FUNCTION "GCS7_SecCtrlMain" : VOID	// FC 60
TITLE = Section Control: Main function
//COPYRIGHT:    (C) 1994 BY  BUHLER AG,  CH-9240 UZWIL  SWITZERLAND
//
//PRODUCT:      GCS7
//
//TITLE:        SECTION CONTROL: MAIN PROGRAM
//
//-------------------------------------------------------------------------
//
//IDENT:        AUTOR:              DEPT:                         DATE:
//
//FB60.3.7      A.Egli              CT3                           07-Mar-2005
//              Move Data: StErrBatch is bit DBX201.0 and not DBX165.0
//FB60.3.6      A.Egli              CT3                           27-Jan-2005
//              Move Data: Compare Job Number, don't use InfSameJobPrevSec 
//FB60.3.5      A.Egli              CT3                           12-Nov-2003
//              Transition to Active: Set JobAc.BatchNo=1 when < 0
//FB60.3.4      A.Egli              CT3                           04-Aug-2003
//              PCRead.Status.StaImmediateStopASW is DBX120.0
//FB60.3.3      A.Egli              CT3                           17-Jul-2003
//              PCDirectControl: ParLineNr is DBW2 and not DBW4
//FB60.3.2      A.Egli              CT3                           12-Jun-2003
//              Wrong lenght copy Line to section
//FB60.3.1      A.Egli              CT3                           14-Mar-2003
//              Code35: Move to any section DB: DBW20=Destination
//              Code22,23: No Transition StEmptying to StWait
//FB60.3.0      A.Egli              CT3                            8-Okt-2002
//              New release
//FB60.2.10     A.Egli              CT3                           18-Mar-2002
//  Send Command only to next section, if InfDataReady=1
//FB60.2.9      A.Egli              CT3                           24-Sept-2001
//  ParStartReleaseTime <=0 : Unlimited time
//FB60.2.8      A.Egli              CT3                           17-Mai-2001
//  Update Last Batch in next section
//FB60.2.7      A.Egli              CT3                            5-Jul-2000
//  Read command from PC only with F_Define 
//FB60.2.6      A.Egli              CT3                           13-Mar-2000
//  Replace DBB73 with DBW72 and DBB9 with DBW8 
//FB60.2E       A.Egli              CT3                           30-Apr-1999
// -Zustandswechsel nach st_emptied: Abfrage DBX117.3 nicht DIX117.3 
//FB60.2D       A.Egli              CT3                           01-Apr-1999
// -Methode 25: Move allways
// -Bei reset Zustandswechsel nach st_emptied (Verbuchung
// -Bei reset kein Zustandswechsel nach  StActive
//FB60.2C       A.Egli              CT3                           22-Jul-98
//               Line-Nr =DBW2
//FB60.2B       A.Egli              AEE6                          14-Mai-98
//               ToASW.InfDataMoved
//FB60.2A       A.Egli              AEE6                          14-Jan-98
//               Update  S5 (Version 2M)
//FB60.1A       A.Egli              AEE6                          16-Jun-96
//               Convert S5 to S7 (Version 2H)
//
//-------------------------------------------------------------------------
//
//PURPOSE:      MANUAL : GCSOSMAN
//
//RESTRICTIONS:
//
//-------------------------------------------------------------------------
//
// CODE of the Methode
//        0    : METHODE CONTROL
//        1    : METHODE DECODER
//        2    : METHODE STEP
//        3    : METHODE STEP_TRANSITION
//        4    : METHODE STATE
//        5    : METHODE MOVE_DATA
//        6    : METHODE NEXT BATCH
//        7    : METHODE O_SECTION
//        9    : METHODE ResultTotal
//        10   : METHODE ResultBatch
//        12   : METHODE PC Direct Control (Diagnose)
//        13   : METHODE WayAdJustTime  
//        25   : METHODE MOVE_DATA Uncondtion
//        35   : METHODE MOVE_DATA any section
//
//ACTUAL DB BY CALL: SECTION  DB
//AUFGESCHALGENER  : SEKTIONS DB
//
//$EJECT
//
//
//
//
//
AUTHOR : EA
FAMILY : GCS7UL
NAME : SEC_MAIN
VERSION : 3.7
VAR_INPUT
  CODE : INT ;	// CODE
END_VAR
VAR_TEMP
  Fault : BOOL ;
  VarLength : INT ;
  tmpByteWrite : INT ;
  SecDBAc : INT ;
  SecDBNext : INT ;
END_VAR
BEGIN
NETWORK
TITLE =
      L     DBNO;
      T     #SecDBAc;
NETWORK
TITLE =  METHODE CONTROL
      L     #CODE;
      L     0;
      <>I;
      JC    aEnd;
// === COMMANDS ==================
      L     DBD 46;	// "SecDB".ToASW.Func
      L     DBD 66;	// "SecDB".ToSSW.Func
      OD;	// 
      T     DBD 46;	// ->"SecDB".ToASW.Func
      L     0;	// 
      ==D;	//   no new commands
      JC    aNoC;
//=== RESET STATUSBIT ======
      L     2#111111;	// ON-COMMAND
      L     DBW 46;	// "SecDB".ToASW.Func[31..16]
      AW;	// 
      INVI;	// 
      L     DBW 120;	// "SecDB".PCRead.Status[15..00]
      AW;	// 
      T     DBW 120;	// ->"SecDB".PCRead.Status[15..00]
// === SET STATUSBIT  ======
      L     2#11111111;	// OFF-COMMAND
      L     DBW 48;	// "SecDB".ToASW.Func[15..00]
      AW;	// 
      L     DBW 120;	// "SecDB".PCRead.Status[15..00]
      OW;	// 
      T     DBW 120;	// -->"SecDB".PCRead.StatusS[15..00]
// 
      A     DBX 121.6;	// "SecDB".PCRead.Status.StaReset
      S     DBX 121.7;	//  "SecDB".PCRead.Status.StaEndOfJob
      A     DBX 48.1;	// "SecDB".ToASW.Func.CmdAbortBacth
      S     DBX 201.0;	// ->"SecDB".JobAc.StaBatch.StaErrBatch
      A     DBX 49.6;	// "SecDB".ToASW.Func.CmdReset
      O     DBX 49.7;	// "SecDB".ToASW.Func.CmdSequenzStop
      O     DBX 48.1;	// "SecDB".ToASW.Func.CmdAbortBacth
      A     DBX 45.7;	//"SecDB".ToASW.InfDataReady [2.10]
      JCN   aNoC;
      CALL  "GCS7_SecCtrlSub" (
           CODE                     := 2);	// SUBROUTINE SEQUENZ_STOP
aNoC: L     0;	// 
      T     DBD 66;	// -> "SecDB".ToSSW.Func
      L     DBW 206;	// "SecDB".JobAc.BatchNo
      L     DBW 168;	// "SecDB".JobNom.BatchNo
      >=I;	// 
      S     DBX 201.3;	// -> "SecDB".JobAc.StaBatch.StaLastBatch
      CALL  "GCS7_SecCtrlSub" (
           CODE                     := 1);	// SUBROUTINE compare
//===Empyting Time =====================================
      AN    DBX 64.2;	//"SecDB".ToSSW.InfPulseTimer
      O     DBX 45.0;	//  "SecDB".ToASW.InfEmptyingTimeEnd
      JC    aE2;	// 
      L     DBW 132;	//"SecDB".PCRead.OutEmptyingTime
      +     1;	// 
      T     DBW 132;	// ->"SecDB".PCRead.OutEmptyingTime
// 
aE2:  A     DBX 62.5;	// "SecDB".ToSSW.InfFeeding
      S     DBX 119.4;	// ->"SecDB".PCRead.Status.StaLoaded
      A     DBX 64.7;	// "SecDB".ToSSW.InfReleaseEmptyingTime
      JC    aX3;	// 
      L     0;	// 
      T     DBW 132;	// "SecDB".PCRead.OutEmptyingTime
aX3:  L     DBW 100;	// "SecDB".PCWrite.ParEmptyingTime
      L     DBW 132;	// "SecDB".PCRead.OutEmptyingTime
      <=I;	// 
      A     DBX 64.7;	//"SecDB".ToSSW.InfReleaseEmptyingTime 
      =     DBX 45.0;	//"SecDB".ToASW.InfEmptyingTimeEnd
      R     DBX 119.4;	// ->"SecDB".PCRead.Status.StaLoaded
      AN    DBX 45.0;	//"SecDB".ToASW.InfEmptyingTimeEnd
      A     DBX 64.7;	// "SecDB".ToSSW.InfReleaseEmptyingTime
      =     DBX 119.6;	// -> "SecDB".PCRead.Status.StaEmptyingTime
//===== F_RESULT =================
      AN    DBX 64.1;	// "SecDB".ToSSW.CmdSendResult
      JC    aCMD;	// 
      AN    DBX 82.1;	// "SecDB".PCWrite.Hsk.Q_Result
      AN    DBX 201.2;	// "SecDB".JobAc.StaBatch.StaRegistrated
      AN    DBX 102.1;	//  "SecDB".PCRead.Hsk.F_Result
      S     DBX 102.1;	//  "SecDB".PCRead.Hsk.F_Result
      S     DBX 41.0;	//  "SecDB".ChangeBit.CBit1 
aCMD: BEU;
aEnd: NOP   0;
NETWORK
TITLE =  METHODE DECODER (Code 1)
      L     #CODE;
      L     1;
      <>I;
      JC    bEnd;
      L     0;
      L     DBB 145;	//  "LineDB".JobWrite.Hsk
      ==I;
      BEC;
      L     DBW 140;	// "LineDB".JobRead.ErrCode   [*1C*]
      L     0;
      <>I;
      BEC;
      L     64;	// Job-Header
      T     DBW 20;	// "LineDB".VarTemp[1] = ObjectNr
      CALL  "GCS7_LineCtrlSub" (
           CODE                     := 1);	// Subroutine block_adr
      OPN   DI [DBW 4];	// -->CALL SECTION-DB[ "LineDB".Para.ParFirstSecDB]
bLop: AN    DIX 44.7;	// "SecDB".ToASW.InfSameJobLineDB
      JC    bNxt;
//  ==== modify datas ===========
      S     DIX 44.0;	// "SecDB".ToASW.CmdModify  
      L     DBD 156;	// "LineDB".JobWrite.Func
      L     DID 46;	// "SecDB".ToASW.Func
      OD;	// 
      T     DID 46;	// --> "SecDB".ToASW.Func
// === Job-Header ==========
      L     DINO;
      T     #SecDBAc;
      CALL  "SYS_Copy_DBtoDB" (
           DBSource                 := DIW 4,
           ByteSource               := 160,
           DBDest                   := #SecDBAc,
           ByteDest                 := 160,
           NoOfByte                 := 40,
           Fault                    := #Fault);	//L_DB / L_DB.DBB160 / SecDB / SecDB.DBB160
// === Telegram: Additional data===
      L     DBW 22;	// "LineDB".VarTemp[2]= VarDWNr
      L     0;	// 
      ==I;	// 
      JC    bEXE;	// 
      L     DIW 12;	// "SecDB".Para.ParSecDataLenNomValue
      T     #VarLength;	// ->VarLenth
      L     DIW 10;	// "SecDB".Para.ParSecDataFirstByte
      L     DIW 14;	// "SecDB".Para.ParSecDataLenAcValue [3.1]
      +I;
      T     #tmpByteWrite;
      CALL  "SYS_Copy_DBtoDB" (
           DBSource                 := DIW 4,
           ByteSource               := DBW 22,
           DBDest                   := #SecDBAc,
           ByteDest                 := #tmpByteWrite,
           NoOfByte                 := #VarLength,
           Fault                    := #Fault);	//L_DB / L_DB.VarDWNr / SecDB
bEXE: AN    DBX 145.1;	//"LineDB".JobWrite.Hsk.F_Execute
      JC    bNxt;
      R     DBX 153.7;	// "LineDB".JobWrite.ObjMask[64]
      L     DBD 146;	// "LineDB".JobWrite.ObjMask[64..01]
      L     DBD 150;	// "LineDB".JobWrite.ObjMask[64..01]
      OD;
      JN    bNxt;
      CDB;
      CALL  "GCS7_SecCtrlSub" (
           CODE                     := 3);	// SUBROUTINE init_section
      CDB;
// -- Call next section
bNxt: L     DIW 8;	// "SecDB".Para.ParNextSecDB
      L     0;	//  
      ==I;	// no next section
      JC    bINI;	// 
      OPN   DI [DIW 8];	// ->CALL SECTION-DB["SecDB".Para.ParNextSecDB]
      JU    bLop;
bINI: R     DBX 153.7;	// "LineDB".JobWrite.ObjMask[64]
      BEU;
bEnd: NOP   0;
NETWORK
TITLE =  METHODE STEP (Code 2 , 22) 
      L     #CODE;
      L     2;
      <>I;
      A(;
      L     #CODE;
      L     22;
      <>I;
      );
      JC    cEnd;
      L     0;
      T     DBW 50;	// "SecDB".ToASW.Transition:=0
      A     DBX 111.0;	//"SecDB".PCRead.Step.StPassive
      JC    cS0;
      A     DBX 111.1;	// "SecDB".PCRead.Step.StWait
      JC    cS1;	// 
      A     DBX 111.2;	//  "SecDB".PCRead.Step.StActive
      JC    cS2;
      A     DBX 111.3;	//  "SecDB".PCRead.Step.StReady
      JC    cS3;
      A     DBX 111.4;	//  "SecDB".PCRead.Step.StEmptying
      JC    cS4;
      A     DBX 111.5;	//  "SecDB".PCRead.Step.StEmptied
      JC    cS5;
      A     DBX 111.6;	//  "SecDB".PCRead.Step.StIdling
      JC    cS6;
      S     DBX 111.0;	// "SecDB".PCRead.Step.StPassive
// === ST_PASSIVE  ========================================
cS0:  A     DBX 45.7;	//"SecDB".ToASW.InfDataReady
      JC    cTx1;	// --> StWait
      JU    cEnd;
// === ST_WAIT ============================================
cS1:  A(;
      L     #CODE;
      L     2;
      ==I;
      );
      A     DBX 121.7;	// "SecDB".PCRead.Status.StaEndOfJob
      AN    DBX 44.5;	// "SecDB".ToASW.InfSameBatchPrevSec
      O     DBX 121.6;	// "SecDB".PCRead.Status.StaReset
      ON    DBX 45.7;	// "SecDB".ToASW.InfDataReady
      JC    cTx5;	// --> StEmpting [2D]
      AN    DBX 116.0;	// es_batchSize
      A     DBX 63.1;	// "SecDB".ToSSW.CmdGotoActive
      JC    cTx2;	// -->  "SecDB".PCRead.Step.StActive
      JU    cEnd;
// ===  "SecDB".PCRead.Step.StActive ==========================================
cS2:  A     DBX 63.2;	// "SecDB".ToSSW.CmdGotoReady
      AN    DBX 44.5;	// "SecDB".ToASW.InfSameBatchPrevSec
      JC    cTx3;	// -->  "SecDB".PCRead.Step.StReady
      L     DBW 72;	//  "SecDB".ToSSW.InNextSecDB
      L     0;	// 
      ==I;	// 
      O     DBX 44.6;	// "SecDB".ToASW.InfSameBatchNextSec
      AN    DBX 44.5;	// "SecDB".ToASW.InfSameBatchPrevSec
      A     DBX 63.3;	//"SecDB".ToSSW.CmdGotoEmptying
      JC    cTx4;	// 
      A     DBX 121.6;	// "SecDB".PCRead.Status.StaReset
      ON    DBX 45.7;	// "SecDB".ToASW.InfDataReady
      JC    cTx5;	// --> StEmpting [2D]
      JU    cEnd;
// ===  "SecDB".PCRead.Step.StReady ==========================================
cS3:  L     DBW 72;	// "SecDB".ToSSW.InNextSecDB
      L     0;	// 
      ==I;	// 
      O     DBX 44.6;	// "SecDB".ToASW.InfSameBatchNextSec
      A     DBX 63.3;	// "SecDB".ToSSW.CmdGotoEmptying
      JC    cTx4;	// -->  "SecDB".PCRead.Step.StEmptying
      A     DBX 121.6;	//  "SecDB".PCRead.Status.StaReset
      ON    DBX 45.7;	//"SecDB".ToASW.InfDataReady
      JC    cTx5;	// --> StEmpting [2D]
      JU    cEnd;
// ===  "SecDB".PCRead.Step.StEmptying =======================================
cS4:  A     DBX 44.5;	// "SecDB".ToASW.InfSameBatchPrevSec
      JC    cTx2;	// -->  "SecDB".PCRead.Step.StActive
      L     DBW 72;	//  "SecDB".ToSSW.InNextSecDB
      L     0;	// 
      ==I;	// 
      O     DBX 44.6;	// "SecDB".ToASW.InfSameBatchNextSec
      A     DBX 63.4;	// "SecDB".ToSSW.CmdGotoEmptied
      JC    cTx5;	// --> StEmptied
      A     DBX 121.6;	//  "SecDB".PCRead.Status.StaReset
      ON    DBX 45.7;	// "SecDB".ToASW.InfDataReady 
      JC    cTx5;	// --> StEmpting [2D]
      JU    cEnd;
// === ST_EMPTIED =======================================
cS5:  A     DBX 44.5;	// "SecDB".ToASW.InfSameBatchPrevSec
      AN    DBX 121.6;	// STA_RESET  [2D]
      JC    cTx2;	// -->  "SecDB".PCRead.Step.StActive
      L     DBW 206;	// "SecDB".JobAc.BatchNo 
      L     DBW 168;	// "SecDB".JobNom.BatchNo
      >=I;	// 
      S     DBX 121.7;	// --> "SecDB".PCRead.Status.StaEndOfJob
      L     0;	// 
      L     DBW 70;	// "SecDB".ToSSW.InPrevSecDB
      ==I;	// 
      A(;
      L     #CODE;
      L     22;
      <>I;
      );
      AN    DBX 121.6;	// "SecDB".PCRead.Status.StaReset 
      AN    DBX 121.7;	// "SecDB".PCRead.Status.StaEndOfJob
      A     DBX 45.7;	// "SecDB".ToASW.InfDataReady
      A     DBX 63.5;	// "SecDB".ToSSW.CmdGotoIdling
      JC    cTx1;	// -->StWait
      A     DBX 121.6;	// "SecDB".PCRead.Status.StaReset [2D]
      ON    DBX 45.7;	//  "SecDB".ToASW.InfDataReady
      AN    DBX 119.3;	//"SecDB".PCRead.Status.StaOnline [2E]
      O     DBX 63.5;	// "SecDB".ToSSW.CmdGotoIdling
      JC    cTx6;	// ->  "SecDB".PCRead.Step.StIdling
      JU    cEnd;
// ===  "SecDB".PCRead.Step.StIdling =======================================
cS6:  A     DBX 45.7;	//  "SecDB".ToASW.InfDataReady
      JC    cTx1;	// --> StWait
      A     DBX 63.6;	//  "SecDB".ToSSW.CmdGotoPassive
      JC    cTx0;	// --> StPassive
      JU    cEnd;
// === TRANSITION =======================================
cTx0: L     2#1;	// --> "SecDB".PCRead.Step.StPassive
      JU    cTra;	// 
cTx1: L     2#10;	// --> "SecDB".PCRead.Step.StWait
      JU    cTra;	// 
cTx2: L     2#100;	// --> "SecDB".PCRead.Step.StActive
      JU    cTra;	// 
cTx3: L     2#1000;	// --> "SecDB".PCRead.Step.StReady
      JU    cTra;	// 
cTx4: L     2#10000;	// --> "SecDB".PCRead.Step.StEmptying
      JU    cTra;	// 
cTx5: L     2#100000;	// --> "SecDB".PCRead.Step.Emptied
      JU    cTra;	// 
cTx6: L     2#1000000;	// -->  "SecDB".PCRead.Step.StIdling
// ==== ALL TRANSITION ==================================
cTra: T     DBW 50;	// --> "SecDB".ToASW.Transition
      BEU;
cEnd: NOP   0;
NETWORK
TITLE =  METHODE TRANSITION_STEP (code 3)
      L     #CODE;
      L     3;
      <>I;
      A(;
      L     #CODE;
      L     23;
      <>I;
      );
      JC    dEnd;
      L     DBW 50;	// "SecDB".ToASW.Transition
      L     0;	// 
      ==I;	// 
      BEC;	// EXIT
      A     DBX 51.0;	// "SecDB".ToASW.Transition.ToPassive
      JC    dTx0;
      A     DBX 51.1;	// "SecDB".ToASW.Transition.ToWait
      JC    dTx1;
      A     DBX 51.2;	// "SecDB".ToASW.Transition.ToActive 
      JC    dTx2;
      A     DBX 51.3;	// "SecDB".ToASW.Transition.ToReady
      JC    dTx3;
      A     DBX 51.4;	// "SecDB".ToASW.Transition.ToEmptying
      JC    dTx4;
      A     DBX 51.5;	// "SecDB".ToASW.Transition.ToEmptied 
      JC    dTx5;
      A     DBX 51.6;	//"SecDB".ToASW.Transition.ToIdling
      JC    dTx6;
      JU    dEnd;
// === TRANSITION_TO_ST_PASSIVE =========================
dTx0: NOP   0;
      JU    dTra;
// === TRANSITION_TO_ST_WAIT ============================
dTx1: R     DBX 63.1;	//  "SecDB".ToSSW.CmdGotoActive 
      R     DBX 64.1;	// "SecDB".ToSSW.CmdSendResult
      A     DBX 111.5;	// "SecDB".PCRead.Step.StEmptied 
      R     DBX 201.0;	// -> "SecDB".JobAc.StaBatch.StaErrBatch
      JU    dTra;
// === TRANSITION_TO_ST_ACTIVE ==========================
dTx2: R     DBX 63.2;	// -> "SecDB".ToSSW.CmdGotoReady
      R     DBX 63.3;	// -> "SecDB".ToSSW.CmdGotoEmptying
      R     DBX 64.1;	// -> "SecDB".ToSSW.CmdSendResult
      L     DBW 206;	// "SecDB".JobAc.BatchNo  [3.5]
      L     1;	//                        [3.5]
      >=I;	//                        [3.5]
      ON    DBX 200.6;	// "SecDB".JobAc.StaBatch.StaEmptyingBatch [3.5]
      JC    dTra;	//                        [3.5]
      T     DBW 206;	// "SecDB".JobAc.BatchNo  [3.5]
      JU    dTra;
// === TRANSITION_TO_ST_READY ==========================
dTx3: R     DBX 63.3;	// -> "SecDB".ToSSW.CmdGotoEmptying
      JU    dTra;
// === TRANSITION_TO_ST_EMPYTYING ======================
dTx4: R     DBX 63.4;	// ->  "SecDB".ToSSW.CmdGotoEmptied
      JU    dTra;
// === TRANSITION_TO_ST_EMPYTIED =======================
dTx5: R     DBX 63.5;	// ->  "SecDB".ToSSW.CmdGotoIdling
      JU    dTra;
// === TRANSITION_TO_StIdling =========================
dTx6: R     DBX 63.6;	// -> "SecDB".ToSSW.CmdGotoPassive
      R     DBX 201.0;	// -> "SecDB".JobAc.StaBatch.StaErrBatch
      R     DBX 200.7;	// -> "SecDB".JobAc.StaBatch.StaScaleRecipeValid
      AN    DBX 121.7;	// [2.8]"SecDB".PCRead.Status.StaEndOfJob 
      JC    dT61;	// [2.8]                
      CALL  "GCS7_SecCtrlSub" (
           CODE                     := 2);	// [2.8] SUBROUTINE SEQUENZ_STOP
dT61: L     0;	// 
      L     DBW 70;	//  "SecDB".ToSSW.InPrevSecDB 
      <>I;	// 
      O(;
      L     #CODE;
      L     23;
      ==I;
      );
      O     DBX 121.7;	// "SecDB".PCRead.Status.StaEndOfJob
      R     DBX 45.7;	// -> "SecDB".ToASW.InfDataReady
      CALL  "GCS7_SecCtrlSub" (
           CODE                     := 7);	// Subroutine TestDone
      AN    DBX 39.0;	// OUTP.JobNotFound
      JC    dTra;	// 
      AN    DBX 102.0;	//  "SecDB".PCRead.Hsk.F_Status 
      S     DBX 201.4;	//"SecDB".JobAc.StaBatch.StaDone
      S     DBX 102.0;	// "SecDB".PCRead.Hsk.F_Status
      S     DBX 41.0;	// "SecDB".ChangeBit.CBit1
dTra: L     DBW 50;	//// "SecDB".ToASW.Transition
      T     DBB 111;	// -->"SecDB".PCRead.Step
      SET;	// 
      S     DBX 41.0;	//  "SecDB".ChangeBit.CBit1
      BEU;
dEnd: NOP   0;
NETWORK
TITLE =  METHODE STATE Code4
      L     #CODE;
      L     4;
      <>I;
      JC    eEnd;
      A     DBX 113.0;	// "SecDB".PCRead.State.StStopped
      JC    eS0;
      A     DBX 113.1;	// "SecDB".PCRead.State.StStarting
      JC    eS1;
      A     DBX 113.2;	// "SecDB".PCRead.State.StStarted 
      JC    eS2;
      A     DBX 113.3;	// "SecDB".PCRead.State.StStopping
      JC    eS3;
      A     DBX 113.5;	// "SecDB".PCRead.State.StFeeding
      JC    eS4;
      S     DBX 113.0;	// "SecDB".PCRead.State.StStopped
// === StStopped  ============
eS0:  AN    DBX 62.0;	// "SecDB".ToSSW.InfStopped
      JC    eT01;	// --> StStarting
      JU    eEnd;	// 
eT01: L     2#10;	// --> StStarting
      JU    eTra;
// === StStarting ============
eS1:  A     DBX 62.2;	// "SecDB".ToSSW.InfStarted
      JC    eT12;	// --> StStarted
      A     DBX 120.0;	// "SecDB".PCRead.Status.StaImmediateStopASW // [3.4]
      O     DBX 62.0;	// "SecDB".ToSSW.InfStopped
      O     DBX 111.6;	// "SecDB".PCRead.Step.StIdling
      JC    eT13;	// -> StStopping
      JU    eEnd;
eT12: L     2#100;	// -> StStarted
      JU    eTra;
eT13: L     2#1000;	// -> StStopping
      JU    eTra;
// === StStarted  ===========
eS2:  A     DBX 120.0;	// "SecDB".PCRead.Status.StaImmediateStopASW
      O     DBX 62.0;	// "SecDB".ToSSW.InfStopped
      JC    eT23;	// --> StStopping
      AN    DBX 62.2;	// "SecDB".ToSSW.InfStarted
      JC    eT21;	// --> StStarting
      A     DBX 62.5;	// "SecDB".ToSSW.InfFeeding
      JC    eT25;	// --> StFeeding
      JU    eEnd;
eT21: L     2#10;	// --> StStarting
      JU    eTra;
eT23: L     2#1000;	// --> StStopping
      JU    eTra;
eT25: L     2#100000;	// --> StFeeding
      JU    eTra;
// ==== STOPPING ==============
eS3:  A     DBX 62.0;	// "SecDB".ToSSW.InfStopped
      JC    eT30;	// -> StStopped
      AN    DBX 120.0;	// "SecDB".PCRead.Status.StaImmediateStopASW
      AN    DBX 62.0;	// "SecDB".ToSSW.InfStopped
      A     DBX 62.2;	// "SecDB".ToSSW.InfStarted
      JC    eT32;	// --> StStarted
      AN    DBX 120.0;	// "SecDB".PCRead.Status.StaImmediateStopASW
      AN    DBX 111.6;	// "SecDB".PCRead.Step.StIdling
      JC    eT32;	// --> StStarting
      JU    eEnd;
eT30: L     2#1;	// --> StStopped
      JU    eTra;
eT32: L     2#100;	// --> StStarted
      JU    eTra;
      L     2#10;	// --> StStarting
      JU    eTra;
// ==== FEEDING  ==============
eS4:  AN    DBX 62.5;	// "SecDB".ToSSW.InfFeeding
      JC    eT52;	// --> StStarted
      JU    eEnd;	// 
eT52: L     2#100;	// --> StStarted
// ==== ALL TRANSITION ========
eTra: T     DBB 113;	// --> "SecDB".PCRead.State
      SET;	// 
      S     DBX 41.0;	// Changebit.CBit1
      BEU;
eEnd: NOP   0;
NETWORK
TITLE =  METHODE MOVE_DATA Code 5,25,35
//Code 35:
//    Section destination=DBW20
      L     #CODE;
      L     5;
      ==I;
      JC    m5;
      L     #CODE;
      L     25;
      ==I;
      JC    m25;
      L     #CODE;
      L     35;
      <>I;
      JC    fEnd;
//Move to section DBW20
      R     DBX 44.2;	//S_DB[n].ToASW.CmdDataMoved
      L     0;
      L     DBW 20;	// "Sec".VarTemp.InOutValue1
      ==I;	// 
      BEC;	// --> no next section
      T     #SecDBNext;
      OPN   DI [#SecDBNext];	// >>>CALL NEXT SECTION-DB["SecDB".ToSSW.InNextSecDB]
      JU    m35;
//====== Move uncondition (Code=25)
m25:  R     DBX 44.2;	//S_DB[n].ToASW.CmdDataMoved
      L     DBW 72;	// "SecDB".ToSSW.InNextSecDB
      L     0;	// 
      ==I;	// 
      BEC;	// --> no next section
      AN    DBX 44.6;	//"SecDB".ToASW.InfSameBatchNextSec
      OPN   DI [DBW 72];	// >>>CALL NEXT SECTION-DB["SecDB".ToSSW.InNextSecDB]
      A     DIX 64.0;	// S_DB[n+1].ToSSW.InfReadyForNewBatch
      AN    DIX 121.3;	// S_DB[n+1].PCRead.Status.StaHold
      A(;
      AN    DIX 102.0;	// S_DB[n+1].PCRead.Hsk.F_Status
      ON    DIX 119.3;	// S_DB[n+1].PCRead.Status.StaOnline
      );
      JC    C3;
      BEU;	// THEN
//=== Move Regular (Code=5)
m5:   R     DBX 44.2;	//S_DB[n].ToASW.CmdDataMoved
      A     DBX 44.6;	// "SecDB".ToASW.InfSameBatchNextSec
      BEC;	//  
      L     DBW 72;	// "SecDB".ToSSW.InNextSecDB
      L     0;	// 
      ==I;	// 
      BEC;	// --> no next section
      OPN   DI [DBW 72];	// >>>CALL NEXT SECTION-DB["SecDB".ToSSW.InNextSecDB]
m35:  A     DBX 201.0;	// S_DB[n+1].JobAc.StaBatch.StaErrBatch
      A     DIX 45.7;	// S_DB[n+1].ToASW.InfDataRead
      BEC;	// 
      A     DIX 201.0;	// S_DB[n+1].JobAc.StaBatch.StaErrBatch       //[3.7]
      A     DIX 45.7;	// S_DB[n+1].ToASW.InfDataReady
      BEC;	// 
      A     DIX 111.0;	// S_DB[n+1].PCRead.Step.StPassive
      O     DIX 111.6;	// S_DB[n+1].PCRead.Step.StIdling
      O     DIX 111.4;	// S_DB[n+1].PCRead.Step.StEmptying
      O     DIX 111.5;	// S_DB[n+1].PCRead.Step.StEmptied
      JC    C2;
      BEU;	// THEN
C2:   A(;	// [3.6]
      L     DID 160;	// [3.6] S_DB[x].JobNom.JobNr
      L     DBD 160;	// [3.6] S_DB[n].JobNom.JobNr
      ==D;	// [3.6] --> InfSameJobPrevSec
      );	// [3.6]
      ON    DIX 45.7;	// S_DB[n+1].ToASW.InfDataReady
      A     DIX 64.0;	// S_DB[n+1].ToSSW.InfReadyForNewBatch
      AN    DIX 121.3;	// S_DB[n+1].PCRead.Status.StaHold
      A(;
      AN    DIX 102.0;	// S_DB[n+1].PCRead.Hsk.F_Status
      ON    DIX 119.3;	// S_DB[n+1].PCRead.Status.StaOnline
      );
      JC    C3;
      BEU;
// ==== MOVE DATA =================
// Copy header
C3:   L     DINO;
      T     #SecDBNext;
      CALL  "SYS_Copy_DBtoDB" (
           DBSource                 := #SecDBAc,
           ByteSource               := 160,
           DBDest                   := #SecDBNext,
           ByteDest                 := 160,
           NoOfByte                 := 80,
           Fault                    := #Fault);	//"SecDB".JobNom.JobNr / Sec[n+1].JobNom.JobNr
//-- copy dynamic datas 
      L     DIW 14;	//Para.ParSecDataLenAcValue
      L     DIW 12;	//Para.ParSecDataLenNomValue
      +I;
      T     #VarLength;
      CALL  "SYS_Copy_DBtoDB" (
           DBSource                 := #SecDBAc,
           ByteSource               := DBW 10,
           DBDest                   := #SecDBNext,
           ByteDest                 := DIW 10,
           NoOfByte                 := #VarLength,
           Fault                    := #Fault);	//Sec[n].Para.ParSecDataFirstByte / Sec[n+1].Para.ParSecDataFirstByte
//-- Copy bin data 
      CALL  "SYS_Copy_DBtoDB" (
           DBSource                 := #SecDBAc,
           ByteSource               := DBW 16,
           DBDest                   := #SecDBNext,
           ByteDest                 := DIW 16,
           NoOfByte                 := DIW 18,
           Fault                    := #Fault);	//Sec[n].Para.ParBinDataFirstByte / Sec[n+1].Para.ParBinDataFirstByte / Sec[n+1].Para.ParBinDataLength
// Init Sec[n+1]
      SET;
      S     DIX 45.7;	//S_DB[n+1].ToASW.InfDataReady 
      S     DIX 44.1;	//S_DB[n+1].ToASW.CmdNewBatch
      S     DBX 44.2;	//S_DB[n].ToASW.CmdDataMoved
      R     DIX 121.6;	//S_DB[n+1].PCRead.Status.StaReset
      R     DIX 121.7;	//S_DB[n+1].PCRead.Status.StaEndOfJob
      R     DIX 64.1;	//S_DB[n+1].ToSSW.CmdSendResult
      AN    DBX 121.0;	//S_DB[n].PCRead.Status.StaImmediateStop   
      R     DIX 121.0;	//S_DB[n+1].PCRead.Status.StaImmediateStop      
      AN    DBX 121.1;	//S_DB[n].PCRead.Status.StaTransferOff
      R     DIX 121.1;	//S_DB[n+1].PCRead.Status.StaTransferOff
      AN    DBX 121.2;	//S_DB[n].PCRead.Status.StaFeedOff
      R     DIX 121.2;	//S_DB[n+1].PCRead.Status.StaFeedOff
      CDB;	// 
      CALL  "GCS7_SecCtrlSub" (
           CODE                     := 1);	//SUBROUTINE compare S_DB[n+1]
      CDB;
      CALL  "GCS7_SecCtrlSub" (
           CODE                     := 1);	//SUBROUTINE compare S_DB[n]
      BEU;
fEnd: NOP   0;
NETWORK
TITLE =  METHODE NEXT_BATCH (code 6)
      L     #CODE;
      L     6;
      <>I;
      JC    gEnd;
      L     DBW 206;	// "SecDB".JobAc.BatchNo
      L     DBW 188;	// "SecDB".JobNom.BatchNoOffset
      >=I;
      JC    gOK;
      T     DBW 206;	// ->"SecDB".JobAc.BatchNo
gOK:  A     DBX 121.7;	// "SecDB".PCRead.Status.StaEndOfJob
      BEC;	// 
//==== start batch ===============
      CALL  "GCS7_SecCtrlSub" (
           CODE                     := 6);	// Subroutine CalcBatchSize
      A     DBX 116.0;	// "SecDB".PCRead.Fault.EsBatchSize
      O     DBX 121.7;	// "SecDB".PCRead.Status.StaEndOfJob
      BEC;
      L     DBD 210;	// "SecDB".JobAc.BatchWeightTarget
      L     DBD 202;	// "SecDB".JobAc.JobWeigth
      +D;	// 
      T     DBD 202;	// ->"SecDB".JobAc.JobWeigth
      L     DBW 206;	//  "SecDB".JobAc.BatchNo
      +     1;	// 
      T     DBW 206;	//  "SecDB".JobAc.BatchNo
      L     0;
      T     DBD 214;	// "SecDB".JobAc.BatchWeightActual
      SET;
      R     DBX 201.1;	//"SecDB".JobAc.StaBatch.StaHandAddReady
      R     DBX 201.2;	//"SecDB".JobAc.StaBatch.StaRegistrated
      L     DBW 206;	//"SecDB".JobAc.BatchNo
      L     DBW 168;	//"SecDB".JobNom.BatchNo
      >=I;	// 
      S     DBX 201.3;	//->"SecDB".JobAc.StaBatch.StaLastBatch 
      SET;	// 
      S     DBX 45.7;	//"SecDB".ToASW.InfDataReady
      S     DBX 44.1;	//"SecDB".ToASW.CmdNewBatch
      CALL  "GCS7_SecCtrlSub" (
           CODE                     := 1);	// SUBROUTINE compare S_DB[n]
      BEU;
gEnd: NOP   0;
NETWORK
TITLE =  METHODE O_SECTION (Code 7)
      L     #CODE;
      L     7;
      <>I;
      JC    hEnd;
      L     DBW 82;	//"SecDB".PCWrite.Hsk
      L     0;
      ==I;
      BEC;
//-- commands --------------
      AN    DBX 83.0;	//"SecDB".PCWrite.Hsk.F_Define [2.7]
      JC    hDef;	// 
      L     DBD 46;	// "SecDB".ToASW.Func
      L     DBD 86;	// "SecDB".PCWrite.Func
      OD;	// 
      T     DBD 46;	// ->"SecDB".ToASW.Func
//--Q_Result----------------
hDef: AN    DBX 82.1;	//"SecDB".PCWrite.Hsk.Q_Result
      JC    hIni;
      S     DBX 201.2;	// "SecDB".JobAc.StaBatch.StaRegistrated 
//---Init Interface---------
hIni: L     DBB 82;	// "SecDB".PCWrite.Hsk.Q_xxxx
      INVI;
      L     DBB 102;	// "SecDB".PCRead.Hsk.F_
      AW;
      T     DBB 102;	// ->Reset "SecDB".PCRead.Hsk.F_xxxx
      L     0;
      T     DBW 82;	// "SecDB".PCWrite.Hsk
      SET;
      S     DBX 41.1;	// "SecDB".ChangeBit.CBit2
      BEU;
hEnd: NOP   0;
NETWORK
TITLE =  METHODE ResultTotal (Code=9)
      L     #CODE;	// )
      L     9;	// )  CODE= KF+9
      <>I;	// )
      JC    iEnd;	// )
      OPN   DI [DBW 4];	//>>call LineDB  DI"SecDB".Para.ParLineDB]
      OPN   DI [DIW 4];	//>>Call 1.SecDB DI["LineDB".Para.ParFirstSecDB]
//Loop over all section
iLop: AN    DIX 45.7;	// S_DB[x].ToASW.InfDataReady
      JC    iNxt;
      L     DID 160;	// S_DB[x].JobNom.JobNr
      L     DBD 160;	// S_DB[n].JobNom.JobNr
      <>D;	// 
      JC    iNxt;
      L     DBD 32;	// "SecDB".VarTemp.InOutValue Input value for registration
      L     DID 202;	// S_DB[x].JobAc.JobWeigth
      +D;	// 
      T     DID 202;	// ->S_DB[x].JobAc.JobWeigth
iNxt: L     0;	// )
      L     DIW 8;	// )   SEC[x].Para.ParNextSecDB
      ==I;	// )
      BEC;	// )
      OPN   DI [DIW 8];	//-->  Call next SecDb  DI["SecDB".Para.ParNextSecDB]
      JU    iLop;
iEnd: NOP   0;
NETWORK
TITLE =  METHODE TotalBatch (Code=10)
      L     #CODE;
      L     10;
      <>I;
      JC    jEnd;
      OPN   DI [DBW 4];	//>>Call LineDB  DI["SecDB".Para.ParLineDB]
      OPN   DI [DIW 4];	//>>Call 1.SecDB DI["LineDB".Para.ParFirstSecDB]
//Loop over all section
jLop: AN    DIX 45.7;	//S_DB[x].ToASW.InfDataReady
      JC    jNxt;
      L     DID 160;	// S_DB[x].JobNom.JobNr
      L     DBD 160;	// S_DB[n].JobNom.JobNr
      <>D;	//  
      JC    jNxt;
      L     DIW 206;	// S_DB[x].JobAc.BatchNo
      L     DBW 206;	// S_DB[n].JobAc.BatchNo
      <>I;	//  
      JC    jNxt;
      L     DBD 32;	// "SecDB".VarTemp.InOutValue  Input value for registration
      L     DID 214;	// JobAc.BatchWeightActual
      +D;	//  
      T     DID 214;	// ->JobAc.BatchWeightActual
jNxt: L     0;	// 
      L     DIW 8;	// SEC[x].Para.ParNextSecDB
      ==I;	// 
      BEC;	// 
      OPN   DI [DIW 8];	//-->Call next SecDb  DI["SecDB".Para.ParNextSecDB]
      JU    jLop;
jEnd: NOP   0;
NETWORK
TITLE =  PC Direct Control (Diagnose) (code= 12)
      L     #CODE;
      L     12;
      <>I;
      JC    kEnd;
      OPN   DI 3;
      L     0;
      L     DIW 42;	// DB3.PC.Hsk
      ==I;	// 
      BEC;	// 
//-- commands --------------
      L     DIW 48;	// DB3.PC.ObjectType
      L     4000;
      <>I;
      BEC;
      L     DIW 50;	// DB3.PC.ObjectNo
      SRW   8;
      L     DBW 2;	// "SecDB".Para.ParLineDB [3.3]
      <>I;
      BEC;
      L     DIB 51;	// DB3.PC.ObjectNo (low byte)
      T     DBW 20;	// "SecDB".VarTemp[1] ==VarSecNr
      CALL  "GCS7_SecCtrlSub" (
           CODE                     := 4);
      L     0;
      T     DBW 22;	// "SecDB".VarTemp[2] == Search_mode=SectionNr
      CALL  "GCS7_SecCtrlSub" (
           CODE                     := 4);	// Subroutine SearchSection
      L     DBW 22;	//"SecDB".VarTemp[2]
      L     0;
      ==I;
      L     20;	// Error code: illegal_object
      JC    ERRO;	// ->illegal section-nr
//--Call Section DB---
      OPN   DB [DBW 22];	// CALL DB["SecDB".VarTemp[2]] = VarSecDB
//  --Commands ------
      AN    DIX 43.0;	// DB3.PC.Hsk.FDefineCmd
      JC    D2;	// 
      L     DID 52;	// DB3..PC.Cmd1
      L     DBD 46;	// "SecDB".ToASW.Func
      OD;	// 
      T     DBD 46;	// "SecDB".ToASW.Func
//  --Parameter ------
D2:   AN    DIX 43.1;	// DB3.PC.Hsk.FDefineCmd
      JC    EXAM;	// 
      L     DIW 58;	// DB3.PC.Value[1]
      T     DBW 90;	// "SecDB".PCWrite.Value1
      L     DIW 60;	// DB3.PC.Value[2]
      T     DBW 92;	// "SecDB".PCWrite.Value2
      L     DIW 62;	// DB3.PC.Value[3]
      T     DBW 94;	// "SecDB".PCWrite.Value3
      L     DIW 64;	// DB3.PC.Value[4]
      T     DBW 96;	// "SecDB".PCWrite.ParWayAdjustTime
      L     DIW 66;	// DB3.PC.Value[5]
      T     DBW 98;	// "SecDB".PCWrite.Value5
      L     DIW 68;	// DB3.PC.Value[6]
      T     DBW 100;	// "SecDB".PCWrite.ParEmptyingTime
//  --Examine ----
EXAM: AN    DIX 43.3;	// DB3.PC.Hsk.FExamine
      JC    DONE;	// 
      L     DBD 90;	// 
      T     DID 58;	// DB3.Value[1..2]
      L     DBD 94;	// 
      T     DID 62;	// DB3.Value[3..4]
      L     DBD 98;	// 
      T     DID 66;	// DB3.Value[5..6]
DONE: L     0;
ERRO: T     "SYS_DirectCtrlDB".PC.ErrCode;	// "SYS_PCControl".PC.ErrCode
      L     0;	// 
      T     "SYS_DirectCtrlDB".PC.Hsk;	// DB3.PC.Hsk
      SET;	//  
      S     "SYS_DirectCtrlDB".ChangeBit.CBit1;	// DB3.ChangeBit.CBit1
      BEU;
kEnd: NOP   0;
NETWORK
TITLE = Methode WayAdJsutTime
      L     #CODE;
      L     13;
      <>I;
      JC    lEnd;
      AN    DBX 64.3;	//"SecDB".ToSSW.CmdNewWay
      JC    lJ1;
      R     DBX 45.1;	//"SecDB".ToASW.InfWayAdjustTimeEnd
      R     DBX 64.3;	//"SecDB".ToSSW.CmdNewWay
      L     0;
      T     DBW 128;	//"SecDB".PCRead.OutWayAdjustTime
lJ1:  A     DBX 45.1;	// "SecDB".ToASW.InfWayAdjustTimeEnd
      BEC;
      AN    "GCS7_Gr_OutTick200ms";
      BEC;
      L     DBW 128;	//"SecDB".PCRead.OutWayAdjustTime
      +     2;
      T     DBW 128;	//"SecDB".PCRead.OutWayAdjustTime
      L     DBW 96;	//"SecDB".PCWrite.ParWayAdjustTime
      >=I;
      S     DBX 45.1;	//"SecDB".ToASW.InfWayAdjustTimeEnd
      BEU;
lEnd: NOP   0;
END_FUNCTION

FUNCTION "GCS7_SecCtrlSub" : VOID	// FC 61
TITLE = Section Control: Subroutines
//COPYRIGHT:    (C) 1994 BY  BUHLER LTD.
//                           CH-9240 UZWIL  SWITZERLAND
//
//PRODUCT:      GCS7
//
//TITLE:        SECTION CONTROL: SUBROUTINE
//
//-------------------------------------------------------------------------
//
//IDENT:        AUTOR:              DEPT:                         DATE:
//
//FC61.2.3      A.Egli              CT3                           08-Mai-2007
//                Modify Batch 
//FC61.2.2      A.Egli              CT3                           12-Aug-2003
//              - Do  not copy StaErrBatch when section is in StWait
//FC61.2.1      A.Egli              CT3                           12-Aug-2003
//              - Compare Prev Section
//FC61.2.0      A.Egli              CT3                            8-Okt-2002
//              - New release
//              - ToASW.InfSameBatchAnyPrevSec 
//              - ToASW.IntSameJobAnyPrevSec 
//FC61.1.5      A.Egli              CT3                            3-Jan-2002
//              Test minimum size : test < not <=
//FC61.1.4      A.Egli              CT3                           14-Apr-2000
//              Test Job active
//FC61.1D       A.Egli              CT3                           11-Juni-1999
//              Calculate number of batch: RND+
//FC61.1C       A.Egli              CT3                           20-Apr-1999
//              Reset EsBatchSizeUpdate by InitSection
//FC61.1B       A.Egli              AEE61                         14-Jan-98
//              Update  to S5 (Version 2G)
//FC61.1A       A.Egli              AEE61                         20-Jun-96
//              Convert to S7 (Version 2F)
//
//-------------------------------------------------------------------------
//
//PURPOSE:      MANUAL : GCSOSMAN
//
//RESTRICTIONS:
//
//-------------------------------------------------------------------------
//
//PARAMETER:
//---------
//  CODE: CODE of the Subroutine
//        KF +1    : SUBROUTINE TEST_MATERIAL
//        KF +2    : SUBROUTINE SEQUENZ_STOP
//        KF +3    : SUBROUTINE INIT_SECTION
//        KF +4    : SUBROUTINE SEARCH_SECTION
//        KF +5    : SUBROUTINE SEARCH_JOB
//        KF +6    : SUBROUTINE CALC_BATCH_SIZE
//        KF +7    : SUBROUTINE TestDone
//
//
AUTHOR : EA
FAMILY : GCS7UL
NAME : SEC_SUBR
VERSION : 2.3
VAR_INPUT
  CODE : INT ;	// CODE
END_VAR
VAR_TEMP
  VarLoop2 : BOOL ;
  VarLastBatch : INT ;
  VarRest : DINT ;
  tmpSameJob : BOOL ;
  tmpSameBatch : BOOL ;
  tmpBatchNo : INT ;
END_VAR
BEGIN
NETWORK
TITLE =
NETWORK
TITLE =  COMPARE (Code 1)
//FLAG IN SUBROUTINE COMPARE: (Batch in previous section and next section)
//==========================
//
      L     #CODE;
      L     1;
      <>I;
      JC    aEND;
      R     DBX 44.3;	// S[n].ToASW.InfSameJobPrevSec
      R     DBX 44.5;	// S[n].ToASW.InfSameBatchPrevSec
      R     DBX 45.2;	// S[n].ToASW.InfSameJobAnyPrevSec
      R     DBX 45.3;	// S[n].ToASW.InfSameBatchAnyPrevSec
      OPN   DI [DBW 4];	//>>Call LineDB  DI["SecDB".Para.ParLineDB]
      OPN   DI [DIW 4];	//>>Call SecDB   DI["LineDB".Para.ParFirstSecDB]
//============================================
//Loop Prev sections
//============================================
pLop: L     DINO;	//Prev Section DB 
      L     DBNO;	//Actual Section DB
      ==I;
      JC    aNXT;
//-- Compare prev. Section
      L     DID 160;	// S[n-1].JobNom.JobNr
      L     DBD 160;	// S[n  ].JobNom.JobNr
      ==D;	// 
      A     DIX 45.7;	// S[n-1].ToASW.InfDataReady
      A     DBX 45.7;	// S[n].ToASW.InfDataReady  [2.1]
      AN    DIX 111.1;	// S[n-1].PCRead.Step.StWait
      =     #tmpSameJob;
      S     DBX 45.2;	// ->S[n].ToASW.InfSameJobAnyPrevSec
      L     DINO;	// Prev Section DB 
      L     DBW 70;	// "SecDB".ToSSW.InPrevSecDB
      ==I;
      A     #tmpSameJob;
      S     DBX 44.3;	// ->S[n].ToASW.InfSameJobPrevSec
//Compare batch
      L     DIW 206;	// S[n-1].JobAc.BatchNo
      L     DBW 206;	// S[n].JobAc.BatchNo
      ==I;	// 
      A     #tmpSameJob;
      =     #tmpSameBatch;
      S     DBX 45.3;	// S[n].ToASW.InfSameBatchAnyPrevSec
      L     DINO;	// Prev Section DB 
      L     DBW 70;	// "SecDB".ToSSW.InPrevSecDB
      ==I;
      A     #tmpSameBatch;
      S     DBX 44.5;	//  )->S[n].ToASW.InfSameBatchPrevSec
//Next 
      L     0;
      L     DIW 8;	// S[i].Para.ParNextSecDB
      ==I;
      JC    aNXT;
      OPN   DI [DIW 8];	//-->  Call next SecDB  DI[Para.ParNextSecDB]
      JU    pLop;
//End Loop Prev sections
//============================================
// Compare next Section
//============================================
aNXT: L     DBW 72;	// "SecDB".ToSSW.InNextSecDB
      L     0;	// 
      <>I;	// 
      A     DBX 45.7;	// "SecDB".ToASW.InfDataReady
      JC    aCM2;	// 
      R     DBX 44.4;	//"SecDB".ToASW.InfSameJobNextSec
      R     DBX 44.6;	//"SecDB".ToASW.InfSameBatchNextSec
      BEU;
aCM2: OPN   DI [DBW 72];	// -> CALL NEXT SECTION DB["SecDB".ToSSW.InNextSecDB]
      L     DID 160;	// S[n+1].JobNom.JobNr
      L     DBD 160;	// "SecDB".JobNom.JobNr
      ==D;
      A     DIX 45.7;	// S[n+1].ToASW.InfDataReady
      AN    DBX 111.1;	// "SecDB".PCRead.Step.StWait
      =     DBX 44.4;	// ->"SecDB".ToASW.InfSameJobNextSec
      L     DIW 206;	// S[n+1].JobAc.BatchNo
      L     DBW 206;	// "SecDB".JobAc.BatchNo
      ==I;
      A     DBX 44.4;	// "SecDB".ToASW.InfSameJobNextSec
      =     DBX 44.6;	// ->S"SecDB".ToASW.InfSameBatchNextSec
      BEU;
aEND: NOP   0;
NETWORK
TITLE =  SEQUENZ_STOP
//1.Scan : Serach last batch
//2.Scan : Set Bit last batch
      L     #CODE;
      L     2;
      <>I;
      JC    bEnd;
      R     #VarLoop2;
      L     0;
      T     #VarLastBatch;
bLo2: OPN   DI [DBW 4];	//>>Call LineDB  DI["SecDB".Para.ParLineDB]
      OPN   DI [DIW 4];	//>>Call SecDB   DI["LineDB".Para.ParFirstSecDB]
//Loop over all section
bLop: L     DID 160;	// S[i].JobNom.JobNr
      L     DBD 160;	// "SecDB".JobNom.JobNr
      <>D;	// 
      JC    bNEQ;	// 
      AN    #VarLoop2;
      JC    bL1;
// ==== LOOP2 =====================
      L     DIW 206;	// S[i].JobAc.BatchNo
      L     #VarLastBatch;
      ==I;	// 
      A     DBX 121.7;	// "SecDB".PCRead.Status.StaEndOfJob
      S     DIX 201.3;	// -> S[i].JobAc.StaBatch.StaLastBatch
      JU    bNEQ;
// === LOOP 1 =====================
bL1:  A     DBX 121.7;	// "SecDB".PCRead.Status.StaEndOfJob 
      S     DIX 121.7;	// ->S[i].PCRead.Status.StaEndOfJob
      L     #VarLastBatch;
      L     DIW 206;	// S[i].JobAc.BatchNo
      >=I;
      JC    bJ1;
      T     #VarLastBatch;
bJ1:  L     DIW 206;	// S[i].JobAc.BatchNo
      L     DBW 206;	// "SecDB".JobAc.BatchNo
      ==I;
      A     DBX 201.0;	// "SecDB".JobAc.StaBatch.StaErrBatch
      AN    DIX 111.1;	//[2.2] S[i].PCRead.StWait
      S     DIX 201.0;	// ->S[i].JobAc.StaBatch.StaErrBatch
bNEQ: L     0;
      L     DIW 8;	// S[i].Para.ParNextSecDB
      ==I;
      JC    bL2;
      OPN   DI [DIW 8];	//-->  Call next SecDB  DI[Para.ParNextSecDB]
      JU    bLop;
//2nd Loop
bL2:  A     #VarLoop2;
      BEC;
      S     #VarLoop2;
      JU    bLo2;
bEnd: NOP   0;
NETWORK
TITLE =  INIT_SECTION
      L     #CODE;
      L     3;
      <>I;
      JC    cEnd;
      S     DBX 45.7;	//"SecDB".ToASW.InfDataReady 
      S     DBX 44.1;	//"SecDB".ToASW.CmdNewBatch
      R     DBX 121.6;	//"SecDB".PCRead.Status.StaReset
      R     DBX 121.7;	//"SecDB".PCRead.Status.StaEndOfJob
      R     DBX 44.3;	//"SecDB".ToASW.InfSameJobPrevSec
      R     DBX 44.5;	//"SecDB".ToASW.InfSameBatchPrevSec
      R     DBX 44.4;	//"SecDB".ToASW.InfSameJobNextSec
      R     DBX 44.6;	//"SecDB".ToASW.InfSameBatchNextSec
      R     DBX 116.0;	//"SecDB".PCRead.Fault.EsBatchSize  [1C]
      L     0;
      T     DBD 202;	//"SecDB".JobAc.JobWeigth
      T     DBW 206;	//"SecDB".JobAc.BatchNo
      L     DBW 200;	//"SecDB".JobAc.StaBatch
      L     2#1000000000000000;
      AW;
      T     DBW 200;	//-->"SecDB".JobAc.StaBatch
      A     DBX 48.1;	// "SecDB".ToASW.Func.CmdAbortBatch
      S     DBX 201.0;	//->"SecDB".JobAc.StaBatch.StaErrBatch
      A     DBX 46.1;	// "SecDB".ToASW.Func.CmdEmptying
      S     DBX 200.6;	//--> "SecDB".JobAc.StaBatch.StaEmptyingBatch
      BEU;
cEnd: NOP   0;
NETWORK
TITLE =  Search section
//SUBROUTINE SEARCH SECTION:
//=======================
//INPUT : ACTUAL DB = Line-DB
//INPUT : LineDB.DBW20: SECTION-NR
//INPUT : LineDB DBW22: search_mode
//             0= Search section with equal section-Nr as DW10
//             1= Search first section with D22.15 ToASW.InfSameJobLineDB==1
//OUTPUT: LineDB DBW22: SECTION-DB
//        0== ILLEGAL SECTION-NR
      L     #CODE;
      L     4;
      <>I;
      JC    dEnd;
      OPN   DI [DBW 4];	//>>Call SecDB DI["LineDB".Para.ParFirstSecDB]
//LOOP:
dLop: L     DIW 2;	//"SecDB".Para.ParSecNr
      L     DBW 20;	//"LineDB".VarTemp[1]= Input.SectionNr.
      ==I;	//  
      AN    DBX 23.0;	//"LineDB".VarTemp[2]= Input.ModeFirstJob
      O;
      A     DBX 23.0;	//"LineDB".VarTemp[2]=Input.ModeFirstJob
      A     DIX 44.7;	//"SecDB".ToASW.InfSameJobLineDB
      JC    dOK;	//->found
      L     DIW 8;	//"SecDB".Para.ParNextSecDB
      L     0;
      ==I;
      JC    dErr;
      OPN   DI [DIW 8];	//--> Call next SecDB  DI["SecDB".Para.ParNextSecDB]
      JU    dLop;
//---End Loop ---
dOK:  L     DINO;	// Actual section DB
dErr: T     DBW 22;	//"LineDB".VarTemp[2] == output Section-DB (0=Not found)
      BEU;
dEnd: NOP   0;
NETWORK
TITLE =  search job
//SUBROUTINE SEARCH JOB:
//=======================
//SEARCH ALL SECTION WITH THE SAME JOB AS IN THE COMMUNICATION DB
//INPUT : ACTUAL DB = COM_DB
//OUTPUT: section-DB D22.15: ToASW.InfSameJobLineDB
//OUTPUT: "LineDB".DBX39.0 (VarTemp[10].0) = Job active
      L     #CODE;
      L     5;
      <>I;
      JC    eEnd;
      R     DBX 39.0;	//LineDB.VarTemp[10] : err_job_active      [1.4] 
//Search Batch number //[2.3]
      L     -1;	//[2.3]
      T     #tmpBatchNo;	//[2.3]
//LOOP all Section:                     //[2.3]
      OPN   DI [DBW 4];	//[2.3]>>Call 1.SecDB DI["LineDB".Para.ParFirstSecDB]
eLp1: L     DBW 154;	//[2.3] "LineDB".JobWrite.SectionDest   
      L     DIW 2;	//[2.3] "SecDB".Para.ParSecNr                  
      ==D;	//[2.3]
      JC    eB1;	//[2.3]
//Call next section                     //[2.3]
      L     DIW 8;	//[2.3] SEC[i].Para.ParNextSecDB      
      L     0;	//[2.3]
      ==I;	//[2.3]
      JC    eL2;	//[2.3]
      OPN   DI [DIW 8];	//Call Next Section //[2.3]
      JU    eLp1;	//[2.3]
eB1:  L     DIW 206;	//[2.3] "SecDB".JobAc.BatchNo     //[2.3]
      T     #tmpBatchNo;	//[2.3]
//---End Loop ---
eL2:  OPN   DI [DBW 4];	//>>Call 1.SecDB DI["LineDB".Para.ParFirstSecDB]
//LOOP:
eLop: SET;
      R     DIX 44.7;	//-->"SecDB".ToASW.InfSameJobLineDB
      A(;
      L     0;
      L     DBW 154;	//"LineDB".JobWrite.SectionDest
      ==I;
      O(;
      L     DIW 2;	//"SecDB".Para.ParSecNr
      ==I;
      );
      O(;	//[2.3]
      L     DIW 206;	//[2.3]  "SecDB".JobAc.BatchNo     //[2.3]
      L     #tmpBatchNo;	//[2.3]
      ==I;	//[2.3]
      A     DBX 145.2;	//[2.3] "LineDB".JobWrite.Hsk.F_Modify  
      );	//[2.3]
      );
      A(;
      L     DID 160;	//"SecDB".JobNom.JobNr
      L     DBD 160;	//"LineDB".JobNom.JobNr
      ==D;
      A     DIX 45.7;	//"SecDB".ToASW.InfDataReady
      O(;
      A     DBX 145.0;	//"LineDB".JobWrite.Hsk.F_Define
      O     DBX 145.1;	// "LineDB".JobWrite.Hsk.F_Execute 
      AN    DIX 45.7;	//"SecDB".ToASW.InfDataReady
      );
      );
      =     DIX 44.7;	//-->"SecDB".ToASW.InfSameJobLineDB
      L     DID 160;	//"SecDB ".JobNom.JobNr                  [1.4]
      L     DBD 160;	//"LineDB".JobNom.JobNr                  [1.4]
      ==D;	//                                       [1.4]
      A     DIX 45.7;	//"SecDB".ToASW.InfDataReady             [1.4]
      S     DBX 39.0;	//-->LineDB.VarTemp[10]= err_job_active [1.4]
//Call next section
      L     DIW 8;	//SEC[i].Para.ParNextSecDB
      L     0;
      ==I;
      BEC;
      OPN   DI [DIW 8];	//DI["SecDB".Para.ParNextSecDBB]
      JU    eLop;
//---End Loop ---
eEnd: NOP   0;
NETWORK
TITLE =  CalcBatchSize (Code 6)
//SUBROUTINE TEST DONE:
//=======================
//SEARCH ALL SECTION WITH THE SAME JOB AS IN THE ACTAUL S_DB
//INPUT : ACTUAL DB = S_DB
//OUTPUT: D19.0: Job not found in a other section
//
//
      L     #CODE;
      L     6;
      <>I;
      JC    fEnd;
      L     DBW 168;	// "SecDB".JobNom.BatchNo
      T     DBW 208;	//->"SecDB".JobAc.BatchNoCal
      L     DBW 186;	// "SecDB".JobNom.BatchMaxPpm
      T     DBW 218;	// "SecDB".JobAc.BatchSizePpm
      L     DBW 168;	//  BatchNoTarget
      L     32767;	// 
      <>I;
      JC    fCAL;	// 
      L     DBD 164;	// "SecDB".JobNom.JobWeight
      L     DBD 202;	// "SecDB".JobAc.JobWeigth
      -D;	//  
      DTR;	// WtRest
      L     DBD 180;	// "SecDB".JobNom.BatchWeight
      DTR;	// 
      /R;	// 
      L     1.000000e+03;	// (promille)
      *R;	// 
      L     DBW 186;	// "SecDB".JobNom.BatchMaxPpm
      DTR;
      /R;
//      L     9.999990e-001
//      +R    
      RND+;	//  NrOfMaxBatch  [1D
      L     DBW 206;	//  "SecDB".JobAc.BatchNo
      +I;	// 
      T     DBW 208;	// ->"SecDB".JobAc.BatchNoCal
      L     DBD 164;	// "SecDB".JobNom.JobWeight
      L     DBD 202;	// "SecDB".JobAc.JobWeigth
      -D;	//  
      DTR;	// WtRest
      L     1.000000e+03;	// (promille)
      *R;	// 
      L     DBD 180;	// "SecDB".JobNom.BatchWeight==100%
      DTR;
      /R;
      RND;
      T     #VarRest;	// WtRest as  ppm
      L     DBW 184;	// "SecDB".JobNom.BatchMinPpm
      <=D;
      A     DBX 201.3;	// "SecDB".JobAc.StaBatch.StaLastBatch
      JC    fDON;	//  -> job done
      <D;	// [Rel 1.5]
      L     #VarRest;	// WtRest as ppm
      JC    fERO;	// ->Fault: EsBatchSize
// Test 1 batches left 
      L     DBW 186;	// "SecDB".JobNom.BatchMaxPpm
      <=D;
      JC    fRST;	// --> Rest
// Test 2 batches left 
      SLD   1;	// 2* batchMaxPc
      <=D;	// 
      JC    fHAF;	// -> batch:= Rest/2
// Maximum Batch
      L     #VarRest;	// WtRestPc as ppm
      L     DBW 186;	// "SecDB".JobNom.BatchMaxPpm
      -D;	// 
      L     DBW 184;	// "SecDB".JobNom.BatchMinPpm
      SLD   1;	// 2*batchMinPc
      >=D;	// 
      L     DBW 186;	// "SecDB".JobNom.BatchMaxPpm
      JC    fSIZ;	// -> batch := "SecDB".JobNom.BatchMaxPpm
// Test 3 batches left
      L     DBW 206;	// "SecDB".JobAc.BatchNo
      +     3;	// 
      T     DBW 208;	// ->"SecDB".JobAc.BatchNoCal
      L     #VarRest;	// 
      DTR;	// 
      L     3.000000e+00;	//   /3
      /R;	// 
      RND;	// VarBatchSizePc
      L     DBW 184;	//  "SecDB".JobNom.BatchMinPpm
      <I;	// 
      JC    fSIZ;	//->Start minimum Size
      TAK;	// 
      JU    fSIZ;	//->Batch Size = Rest/3
fHAF: L     #VarRest;
      SSD   1;	//  /2
      L     DBW 184;	//  "SecDB".JobNom.BatchMinPpm
      >=I;
      TAK;
      JC    fSIZ;	// -> Batch Size = Rest/2
      JU    fERO;
//== Error =====================
fERO: T     DBW 218;	//"SecDB".JobAc.BatchSizePpm
      A     DBX 47.7;	// "SecDB".ToASW.Func.CmdAcceptSize
      JC    fSIZ;	// 
      AN    DBX 116.0;	// "SecDB".PCRead.Fault.EsBatchSize
      S     DBX 116.0;	// -> "SecDB".PCRead.Fault.EsBatchSize
      S     DBX 48.3;	// ->"SecDB".ToASW.Func.CmdHornOn
      JU    fCAL;
// === Start Batch ===============
//Error batch size
fDON: R     DBX 116.0;	// -> "SecDB".PCRead.Fault.EsBatchSize  
      S     DBX 121.7;	// ->"SecDB".PCRead.Status.StaEndOfJob
      L     DBW 206;	//  "SecDB".JobAc.BatchNo 
      T     DBW 208;	// ->"SecDB".JobAc.BatchNoCal
      BEU;
//Last Batch
fRST: S     DBX 201.3;	//->"SecDB".JobAc.StaBatch.StaLastBatch
      L     #VarRest;	//var_WtRestPc
fSIZ: T     DBW 218;	//-->"SecDB".JobAc.BatchSizePpm
      R     DBX 116.0;	//-> "SecDB".PCRead.Fault.EsBatchSize
fCAL: L     DBW 218;	//"SecDB".JobAc.BatchSizePpm
      DTR;	// 
      L     DBD 180;	// "SecDB".JobNom.BatchWeight
      DTR;	// 
      *R;	// 
      L     1.000000e+03;	// [1/1000]
      /R;	// 
      RND;	// 
      T     DBD 210;	// ->"SecDB".JobAc.BatchWeigthTarget
      BEU;
fEnd: NOP   0;
NETWORK
TITLE =  TestDone Code 7)
      L     #CODE;	// 
      L     7;	// 
      <>I;	// 
      JC    gEnd;	// 
      S     DBX 39.0;	// outp_NotFound
      OPN   DI [DBW 4];	//>>call LineDB  DI["SecDB".Para.ParLineDB]
      OPN   DI [DIW 4];	//>>Call 1.SecDB DI["LineDB".Para.ParFirstSecDB]
//Loop over all section
gLop: L     DID 160;	// SecDB[i].JobNom.JobNr
      L     DBD 160;	// "SecDB".JobNom.JobNr
      <>D;	// 
      ON    DIX 45.7;	// "SecDB".ToASW.InfDataReady
      JC    gNeq;	// 
      L     DINO;	// SecDB[i]
      L     DBNO;	// SecDB
      <>I;	// 
      R     DBX 39.0;	// outp_NotFound
gNeq: L     DIW 8;	// SecDB[i].Para.ParNextSecDB
      L     0;	// 
      ==I;	// 
      BEC;	// 
//-->Call next SecDB  DI["SecDB".Para.ParNextSecDB]
      OPN   DI [DIW 8];
      JU    gLop;
//---End Loop ---
gEnd: NOP   0;
NETWORK
TITLE =
END_FUNCTION

FUNCTION "GCS7_BinCtrlMain" : VOID	// FC 66
TITLE = Bin Control: Main Routines
//COPYRIGHT:    (C) 1994 BY  BUHLER LTD.
//                           CH-9240 UZWIL  SWITZERLAND
//
//PRODUCT:      GCS7
//
//TITLE:        BIN CONTROL: MAIN PROGRAM
//
//-------------------------------------------------------------------------
//
//IDENT:        AUTOR:              DEPT:                         DATE:
//FC66.3.4      A.Egli              CT3                           05-Jul-2004
//              PCRead.Status.StaListNotUsed 1->0: Change to first bin 
//FC66.3.3      A.Egli              CT3                           02-Jul-2004
//              Methode InitData: Check is bin is active
//FC66.3.2      A.Egli              CT3                           04-Jun-2004
//              Deselect active bin when list is not used 
//FC66.3.1      A.Egli              CT3                           04-Mai-2004
//              Set change bit when registering PrevJob 
//FC66.3.0      A.Egli              CT3                           07-Oct-2002
//              New release 
//FC66.2.1      A.Egli              CT3                           22-Mai-2002
//              Init Data: Change directlty to first OK ingredient    
//FC66.2.0      A.Egli              CT3                           18-Jan-2002
//              ToASW.OutJobChange: Dont't result to bins of the old job
//FC66.1.7      A.Egli              CT3                            7-Jun-2001
//              Reset InfPreselect, if Bin is allredy active
//FC66.1.6      A.Egli              CT3                            8-Feb-2001
//              Reset InfEmptyRecipe in Methode "Decoder"
//FC66.1.5      A.Egli              CT3                           29-Jun-2000
//              CmdNext 
//FC66.1.4      A.Egli              CT3                           05-Mai-2000
//              ErrObject 
//FC66.1D       A.Egli              AEE6                          14-Mai-98
//              Update  to S5 (Rel 2B)
//FC66.1C       A.Egli              AEE6                          30-Mar-98
//              Update  to S5 (Rel 2A)
//FC66.1B       A.Egli              AEE6                          14-Jan-98
//              Update  to S5 (Rel 1N)
//FC66.1A       A.Egli              AEE6                          24-Jun-96
//              Convert from S5 (Rel 1H)
//
//-------------------------------------------------------------------------
//
//PURPOSE:      MANUAL : BINMAN
//
//RESTRICTIONS:
//
//-------------------------------------------------------------------------
//
//
AUTHOR : EA
FAMILY : GCS90UL
NAME : BIN_MAIN
VERSION : 3.4
VAR_INPUT
  CODE : INT ;	// CODE
END_VAR
VAR_TEMP
  VarLenRecipe : INT ;
  VarSecDB : INT ;
  VarLineDB : INT ;
  varBinDB : INT ;
  VarInByteRecipe : INT ;	//Position Recipe in Line-DB
  VarError : BOOL ;
  VarNewJob : BOOL ;
  VarAddrBin : DWORD ;
  VarAddrBinIdx : DWORD ;
  VarAddrPointer : DWORD ;
  VarAddrIdx : DWORD ;
  VarCnt : INT ;
  VarNoLL : BOOL ;
  VarNoHL : BOOL ;
  VarAddElement : DWORD ;
  VarLenBinBit : DINT ;
  VarIngrIdx : INT ;
  VarCntBin : INT ;
  VarBinNr : INT ;
  VarCentBinIdx : INT ;
  VarAddrCentBin : DWORD ;
  VarCentLenBinBit : DINT ;
END_VAR
BEGIN
NETWORK
TITLE =
//CODE: 
//        0    : METHODE CONTROL
//        1    : METHODE DECODER
//        2    : METHODE INIT DATA
//        7    : METHODE O_BIN
//        8    : METHODE TEST_RECIPE
//       10    : METHODE TOTALIZER
//       11    : METHODE JOBCHANGE
//       18    : METHODE TEST_RECIPE: Test Last Bin Active
//
//ACTUAL DB BY CALL: DB Bin control
//
//
//=========================================
//Methode CONTROL: +0
//---------------
//Input:
//  Actual DB Bin_Contol
//=========================================
//
//Methode DECODER: Code=1
//---------------
//Input:
//  Actual DB Bin_Contol
//
//=========================================
//
//Methode Init Data: Code=2
//----------------------------
//Input:
//  Actual DB Bin_Contol
//
//=========================================
//
//Methode PCDirectControl (Diagnose) : Code=7
//----------------------------
//Input:
//  Actual DB Bin_Contol
//
//=========================================
//Methode Test_Recipe: Code=+8
//------------------------------
//Input:
//  Actual DB Bin_Contol
//  Input: DBW20="BinDB".VarTemp.InValue     = Source Recipe DBNr
//Output:
//  DBX   39.0                  //"BinDB".VarTemp.Value10.tmpBinNotFound1 
//  DBX   39.1                  //"BinDB".VarTemp.Value10.tmpLevelFault
//  DBX   39.2                  //"BinDB".VarTemp.Value10.tmpBinNotFound2
//  DBX   39.3                  //"BinDB".VarTemp.Value10.tmpEmptyRecipe
//  DBX   39.4                  //"BinDB".VarTemp.Value10.tmpFull
//
//
//=========================================
//Methode Totalizer: Code=+10
//------------------------------
//Input:
//Output:
//  DBD64    0            // "BinDB".ToSSW.WeightTotal
//
//
      L     DBW 10;	// "BinDB".Para.ParNoOfBytePerBin
      SLD   3;
      T     #VarLenBinBit;
NETWORK
TITLE =  Length Test
      L     DBW 10;	// "BinDB".Para.ParNoOfBytePerBin
      L     DBW 12;	// "BinDB".Para.ParNoOfBin
      *I;
      L     DBW 8;	// "BinDB".Para.ParByteFirstBin
      +I;
      L     DBLG;	//  Actual DB Lenght
      >I;
      JCN   aEnd;
      S     DBX 103.3;	//  -->"BinDB".PCRead.Fault.EsCfgFault
      S     DBX 103.1;	//  -->"BinDB".PCRead.Fault.EsLevelFault
      BEU;
aEnd: NOP   0;
NETWORK
TITLE =  Methode Control (Part.1)
      L     #CODE;
      L     0;
      <>I;
      JC    C1;
      R     DBX 39.7;	// "BinDB".VarTemp.Value10.Flag7
      AN    DBX 105.5;	//PCRead.Status.StaListNotUsed        [3.4]
      A     DBX 38.0;	//VarTmp.Value10.Flag8                [3.4]
      AN    DBX 43.1;	//"BinDB".ToASW.InfPreselect          [3.4]
      S     DBX 61.0;	//-> "BinDB".VarCommand.CmdFirst      [3.4]
//[3.2]-->             
//Deselect active bin when list is not active
      A     DBX 105.5;	//PCRead.Status.StaListNotUsed
      FP    DBX 38.0;	//VarTmp.Value10.Flag8
      JCN   dNAC;
//    ) Subroutine: Deselect all
      CALL  "GCS7_BinCtrlSub" (
           CODE                     := 4);
dNAC: NOP   0;
//<--[3.2]
//   **** commands *****************
      A     DBX 103.2;	// "BinDB".PCRead.Fault.EsNoNextBin
      =     DBX 60.4;	// "BinDB".VarCommand.InfFlagEsNoNextBin
//  --Rel S5.1I
      AN    DBX 60.6;	// "BinDB".VarCommand.InfEmptyRecipe
      AN    DBX 60.7;	// "BinDB".VarCommand.CmdNewValue
      JC    b0X0;
      CALL  "GCS7_BinCtrlMain" (
           CODE                     := 18);	// Test Recipe/ Test Last Bin Active     [3.0]
//  --End S5.1I
b0X0: A     DBX 62.5;	// "BinDB".ToSSW.CmdFirst
      R     DBX 62.5;	// "BinDB".ToSSW.CmdFirst
      S     DBX 61.0;	//-> "BinDB".VarCommand.CmdFirst
      A     DBX 62.6;	// "BinDB".ToSSW.CmdNext
      R     DBX 62.6;	// "BinDB".ToSSW.CmdNext
      S     DBX 61.1;	//->"BinDB".VarCommand.CmdNext
//  --Rel S5.1L
      AN    DBX 105.2;	// "BinDB".PCRead.Status.StaSpecialBin
      O     DBX 7.0;	// "BinDB".Para.ParTypeDef.ParBlend 
      JC    b0OK;
      OPN   DI [DBW 4];	//   DB["BinDB".Para.ParSecDB]
      L     DBW 18;	// "BinDB".Para.ParNoOfIngr
      +     -1;
      L     DBW 16;	// "BinDB".Para.ParNoOfBytePerIngr
      *D;
      L     DBW 14;	// "BinDB".Para.ParByteRecipeMemory
      +D;
      +     L#6;	//    WeightTotal + StatusRec
      SLD   3;	//    
      T     #VarAddrPointer;	//   -->Address recipe
      L     DIW [#VarAddrPointer];	//   specal bin form recipe
      L     DBW 50;	// "BinDB".ToASW.BinPreselected
      <>I;
      O;
      A     DBX 105.2;	// "BinDB".PCRead.Status.StaSpecialBin 
      AN    DBX 61.2;	// "BinDB".VarCommand.VarSpecialBin
      S     DBX 61.1;	//->"BinDB".VarCommand.CmdNext  //  1.5
//  --End S5.1L
b0OK: AN    DBX 105.2;	// "BinDB".PCRead.Status.StaSpecialBin
      A     DBX 61.2;	// "BinDB".VarCommand.VarSpecialBin  
      S     DBX 61.1;	//->"BinDB".VarCommand.CmdNext
      AN    DBX 105.2;	// "BinDB".PCRead.Status.StaSpecialBin
      A     DBX 61.2;	// "BinDB".VarCommand.VarSpecialBin
      S     DBX 60.5;	//  --> "BinDB".VarCommand.InfBinNotInRecipe
      A     DBX 105.2;	// "BinDB".PCRead.Status.StaSpecialBin
      =     DBX 61.2;	// "BinDB".VarCommand.VarSpecialBin
//   === NO Ingredient in Recipe ===
      A     DBX 60.6;	// "BinDB".VarCommand.InfEmptyRecipe
      AN    DBX 105.2;	// "BinDB".PCRead.Status.StaSpecialBin
      A     DBX 43.0;	// "BinDB".ToASW.InfActive
      AN    DBX 43.2;	// "BinDB".ToASW.InfDeselect
      JCN   b000;
//     Subroutine: Deselect all
      CALL  "GCS7_BinCtrlSub" (
           CODE                     := 4);
//   ****Test bin-status ************
b000: CALL  "GCS7_BinCtrlSub" (
           CODE                     := 0);	//   Subroutine Test bin status
//   **** var_new_value  ************
      AN    DBX 60.7;	// "BinDB".VarCommand.CmdNewValue
      JC    bCD2;
      R     DBX 60.7;	// "BinDB".VarCommand.CmdNewValue
      OPN   DI [DBW 4];	//   DB[ParSectionDB]
      L     DBW 14;	// "BinDB".Para.ParByteRecipeMemory 
      SLW   3;	//   
      LAR1;
      T     #VarAddrPointer;	// 
      L     DID [AR1,P#2.0];	// S_DB.L01Rcv1.WeightTotal
      T     DBD 78;	// --> "BinDB".ToSSW.WeightTotalNom
      T     DBD 120;	// -->"BinDB".PCRead.WeightTotalRec
      L     DIW [AR1,P#0.0];	//  S_DB.L01Rcv1.StatusRec
      T     DBW 118;	// --> "BinDB".PCRead.StatusRec
//   ==== Transport ===========================================
      A     DBX 7.0;	// "BinDB".Para.ParTypeDef.ParBlend 
      JC    bBLE;
      L     2#10;	//   Mode Read Value
      T     DBW 20;	// "BinDB".VarTemp.InValue
      CALL  "GCS7_BinCtrlSub" (
           CODE                     := 13);	//   Subroutine ReadBlendRecipe
      L     DBW 48;	// "BinDB".ToASW.BinActual
      AN    DBX 43.1;	// "BinDB".ToASW.InfPreselect
      JC    bX1;	//   
      L     DBW 50;	// "BinDB".ToASW.BinPreselected
bX1:  T     DBW 20;	// "BinDB".VarTemp.InValue
      CALL  "GCS7_BinCtrlSub" (
           CODE                     := 10);	//  Subroutine Position Ingr.
      AN    DBX 39.0;	// "BinDB".VarTemp10.tmpBinNotFound1 
      JC    bCD2;
      S     DBX 61.0;	// "BinDB".VarCommand.CmdFirst
      S     DBX 60.5;	// "BinDB".VarCommand.InfBinNotInRecipe
      JU    bCD2;
      JU    C0P2;	//->Part 2
//   ==== BLEND ===========================================
bBLE: CALL  "GCS7_BinCtrlSub" (
           CODE                     := 4);	//   Subroutine Deselect all
      L     2#1;	//   CODE= Preselect
      T     DBW 20;	// "BinDB".VarTemp.InValue
      CALL  "GCS7_BinCtrlSub" (
           CODE                     := 13);	//   Subroutine Read Blend Recipe
      CALL  "GCS7_BinCtrlSub" (
           CODE                     := 0);	//   Subroutine Test Bin Status
      L     2#10;	//   CODE= Read Value
      T     DBW 20;	// "BinDB".VarTemp.InValue
      AN    DBX 43.1;	// "BinDB".ToASW.InfPreselect
      AN    DBX 43.2;	// "BinDB".ToASW.InfDeselect
      JCN   bCD2;
//   === Test wa adjust time ===
      CALL  "GCS7_BinCtrlSub" (
           CODE                     := 13);	//   Subroutine Read Blend Recipe
bCD2: NOP   0;
//  === F_RESULT =================
      AN    DBX 62.1;	// "BinDB".ToSSW.CmdSendResult
      JC    bCD4;	//     
      AN    DBX 105.3;	// "BinDB".PCRead.Status.StaRegistrated
      AN    DBX 82.1;	// "BinDB".PCWrite.Hsk.Q_Result
      AN    DBX 94.1;	// "BinDB".PCRead.Hsk.F_Result
      S     DBX 94.1;	// "BinDB".PCRead.Hsk.F_Result
      S     DBX 41.0;	// "BinDB".ChangeBit.CBit1
//   === READ VALUE BEND ============
bCD4: AN    DBX 7.0;	// "BinDB".Para.ParTypeDef.ParBlend
      AN    DBX 7.3;	// "BinDB".Para.ParTypeDef.ParWithTargetValue
      ON    DBX 62.7;	// "BinDB".ToSSW.CmdReadNewValue
      JC    C0P2;	//   
      R     DBX 62.7;	// "BinDB".ToSSW.CmdReadNewValue
      L     2#10;	//   code Read Value/read Bin
      T     DBW 20;	// "BinDB".VarTemp.InValue
      CALL  "GCS7_BinCtrlSub" (
           CODE                     := 13);	//   Subroutine Read Blend Recipe
NETWORK
TITLE =  Methode Control Code 0 (Part.2)
// === Find next ingredient ====
C0P2: AN    DBX 60.6;	// "BinDB".VarCommand.InfEmptyRecipe
      AN    DBX 60.5;	// "BinDB".VarCommand.InfBinNotInRecip
      A     DBX 43.0;	// "BinDB".ToASW.InfActive  
      AN    DBX 103.1;	// "BinDB".PCRead.Fault.EsLevelFault 
      R     DBX 103.2;	// "BinDB".PCRead.Fault.EsNoNextBin
      A     DBX 60.5;	// "BinDB".VarCommand.InfBinNotInRecipe
      S     DBX 61.1;	//   )-> "BinDB".VarCommand.CmdNext
//   ---Transport --------------------
      A     DBX 7.0;	// "BinDB".Para.ParTypeDef.ParBlend
      JC    cBLN;
      A     DBX 61.0;	// "BinDB".VarCommand.CmdFirst
      R     DBX 61.0;	// "BinDB".VarCommand.CmdFirst
      JC    cBI1;	//  --> first bin
      A     DBX 61.1;	// "BinDB".VarCommand.CmdNext 
      JC    cFND;
      AN    DBX 103.0;	// "BinDB".PCRead.Fault.EsLevelWarning 
      AN    DBX 103.1;	// "BinDB".PCRead.Fault.EsLevelFault
      JC    cCD1;
      L     DBW 48;	// "BinDB".ToASW.BinActual
      T     DBW 20;	// "BinDB".VarTemp.InValue    
      CALL  "GCS7_BinCtrlSub" (
           CODE                     := 2);	//   Subroutine Read bin
      A     DBX 39.0;	// "BinDB".VarTemp10.tmpBinNotFound1
      JC    cFND;	//   
      AN    DBX 24.0;	//   bin[n].InfLocked
      AN    DBX 24.1;	//   bin[n].InfLevelFault
      AN    DBX 60.5;	// "BinDB".VarCommand.InfBinNotInRecipe
      JC    cCD1;	//   
cFND: R     DBX 61.1;	// "BinDB".VarCommand.CmdNext
      R     DBX 38.7;	//   var_second_loop
      L     DBW 48;	// "BinDB".ToASW.BinActual  
      T     DBW 20;	// "BinDB".VarTemp.InValue
      CALL  "GCS7_BinCtrlSub" (
           CODE                     := 10);	//   Subroutine Position Ingr.
      A     DBX 39.0;	// "BinDB".VarTemp10.tmpBinNotFound1
      JC    cF1;
//   ---- Read Next ----------------
cNXT: CALL  "GCS7_BinCtrlSub" (
           CODE                     := 12);	//   Subroutine Read next
      JU    cTST;
//   ---- Read first ---------------
cF1:  A     DBX 38.7;	//   var_second_loop
      JC    cNOB;	//   
cBI1: S     DBX 38.7;	//   var_second_loop
      CALL  "GCS7_BinCtrlSub" (
           CODE                     := 11);	//   Subroutine ReadFirst
cTST: A     DBX 39.0;	// "BinDB".VarTemp10.tmpBinNotFound1  
      AN    DBX 7.1;	// "BinDB".Para.ParTypeDef.ParLoopIngr
      JC    cNOB;	//   
      A     DBX 39.0;	// "BinDB".VarTemp10.tmpBinNotFound1
      JC    cF1;
//   ---- Test Level ---------------
      CALL  "GCS7_BinCtrlSub" (
           CODE                     := 2);	//   Subroutine Read bin
      A     DBX 39.0;	// "BinDB".VarTemp10.tmpBinNotFound1
      JC    cNXT;	//   
      A     DBX 24.0;	//   bin[n].InfLocked
      O     DBX 24.1;	//   bin[n].InfLevelFault
      A(;
      AN    DBX 60.5;	// "BinDB".VarCommand.InfBinNotInRecipe
      ON    DBX 103.2;	// "BinDB".PCRead.Fault.EsNoNextBin
      AN    DBX 105.2;	// "BinDB".PCRead.Status.StaSpecialBin
      );
      JC    cNXT;
//   ---- Preselect bin -----------
      R     DBX 60.5;	// "BinDB".VarCommand.InfBinNotInRecipe
      A     DBX 103.2;	// "BinDB".PCRead.Fault.EsNoNextBin
      R     DBX 103.2;	//-> "BinDB".PCRead.Fault.EsNoNextBin
      S     DBX 41.0;	//->  "BinDB".ChangeBit.CBit1
//    ) Subroutine: Deselect all
      CALL  "GCS7_BinCtrlSub" (
           CODE                     := 4);
      L     DBW 20;	//    var_bin_nr
      T     DBW 50;	// "BinDB".ToASW.BinPreselected
      AN    DBX 25.0;	// "BinDB".VarTemp.Bin.InfActiveBin [1D]
      O     DBX 25.2;	// "BinDB".VarTemp.Bin.InfDeselect
      S     DBX 25.1;	// "BinDB".VarTemp.Bin.InfPreselect
      R     DBX 25.2;	// "BinDB".VarTemp.Bin.InfDeselect
      A     DBX 25.0;	// "BinDB".VarTemp.Bin.InfActiveBin[1.7]
      R     DBX 25.1;	// "BinDB".VarTemp.Bin.InfPreselect [1.7]
//   Subroutine: Store bin
      CALL  "GCS7_BinCtrlSub" (
           CODE                     := 3);
      JU    cCD2;
//   (====END NEXT INGR.TRANSPORT===)
cNOB: AN    DBX 103.2;	// "BinDB".PCRead.Fault.EsNoNextBin
      S     DBX 103.2;	//   ==> "BinDB".PCRead.Fault.EsNoNextBin
      AN    DBX 60.4;	// "BinDB".VarCommand.InfFlagEsNoNextBin 
      S     DBX 41.0;	// "BinDB".ChangeBit.CBit
      JU    cCD1;
//   ====READ RECIPE BLEND ==========
//   ---Blend --------------------
cBLN: AN    DBX 61.0;	// "BinDB".VarCommand.CmdFirst
      JC    cCD1;
      R     DBX 61.0;	// "BinDB".VarCommand.CmdFirst
//   Subroutine: Deselect all
      CALL  "GCS7_BinCtrlSub" (
           CODE                     := 4);
      L     2#1;	//   code Read Bin
      T     DBW 20;	// "BinDB".VarTemp.InValue
      JCN   cCD2;
//   Subroutine: Read Blend Recipe
      CALL  "GCS7_BinCtrlSub" (
           CODE                     := 13);
//    Subroutine: Test Bin Status
cCD2: CALL  "GCS7_BinCtrlSub" (
           CODE                     := 0);
cCD1: NOP   0;
//   **** Seclect New Bin ***********
      A     DBX 63.1;	// "BinDB".ToSSW.CmdReadyForSelect 
      A     DBX 43.1;	// "BinDB".ToASW.InfPreselect 
      O;	//   
      A     DBX 63.2;	// "BinDB".ToSSW.CmdReadyForDeselect
      A     DBX 43.2;	// "BinDB".ToASW.InfDeselect
      JC    cBNS;	//   
      JU    cCD3;
//   -- select bins ----------
//   Subroutine: Modify_bin
cBNS: CALL  "GCS7_BinCtrlSub" (
           CODE                     := 5);
      L     2#10;	// Read Value
      T     DBW 20;	// "BinDB".VarTemp.InValue
//   Subroutine: Read Blend Recipe
      CALL  "GCS7_BinCtrlSub" (
           CODE                     := 13);
//   Subroutine: Test Bin Status
      CALL  "GCS7_BinCtrlSub" (
           CODE                     := 0);	//   Subroutine Test Bin Status
//   ***** REGISTERING **********
cCD3: AN    DBX 43.1;	// "BinDB".ToASW.InfPreselect  [2.0]
      AN    DBX 43.2;	// "BinDB".ToASW.InfDeselect   [2.0]
      R     DBX 43.6;	// "BinDB".ToASW.OutJobChange  [2.0]
      A     DBX 43.6;	// "BinDB".ToASW.OutJobChange  [2.0]
      AN    DBX 62.1;	// "BinDB".ToSSW.CmdSendResult [2.0]
      AN    DBX 94.1;	// "BinDB".PCRead.Hsk.F_Result  [2.0]
      O     DBX 7.0;	// "BinDB".Para.ParTypeDef.ParBlend
      JC    cCD5;	//   
      L     DBD 64;	// "BinDB".ToSSW.WeightTotal
      L     DBD 44;	// "BinDB".ToASW.VarTaraWeight
      -D;	//   
      JP    cRES;	//   
      JU    cCD5;	//   
cRES: L     DBW 48;	// "BinDB".ToASW.BinActual 
      T     DBW 20;	// "BinDB".VarTemp.InValue 
      CALL  "GCS7_BinCtrlSub" (
           CODE                     := 2);	//   Subroutine read bin
      A     DBX 39.0;	// "BinDB".VarTemp.Value10.tmpBinNotFound1 
      JC    cCD5;	//    
      L     DBD 64;	// "BinDB".ToSSW.WeightTotal
      L     DBD 44;	// "BinDB".ToASW.VarTaraWeight 
      -D;	//   
      L     DBD 28;	// "BinDB".VarTemp.Bin.WeightActual
      +D;	//   
      T     DBD 28;	// "BinDB".VarTemp.Bin.WeightActual 
      L     DBD 64;	// "BinDB".ToSSW.WeightTotal
      T     DBD 44;	//->"BinDB".ToASW.VarTaraWeight
      CALL  "GCS7_BinCtrlSub" (
           CODE                     := 3);	//  Subroutine Store bin
//  --Emptying time ----------
cCD5: AN    DBX 63.4;	// "BinDB".ToSSW.CmdPulseTimer
      O     DBX 43.7;	// "BinDB".ToASW.InfEmptyingEnd
      JC    cX1;	//   
      L     DBW 116;	// "BinDB".PCRead.OutEmptyingTime
      +     -1;	//   
      T     DBW 116;	//->"BinDB".PCRead.OutEmptyingTime
cX1:  A     DBX 63.7;	// "BinDB".ToSSW.InfReleaseEmptyingTime
      JC    cX3;	//   
      L     DBW 92;	// "BinDB".PCWrite.ParEmptyingTime
      L     DBW 52;	// "BinDB".ToASW.OutEmptyingTimeBin
      <=I;
      JC    xJ6;
      TAK;
xJ6:  T     DBW 116;	// "BinDB".PCRead.OutEmptyingTime
cX3:  L     DBW 116;	// "BinDB".PCRead.OutEmptyingTime
      L     0;
      <=I;
      A     DBX 63.7;	// "BinDB".ToSSW.InfReleaseEmptyingTime
      =     DBX 43.7;	// "BinDB".ToASW.InfEmptyingEnd 
      R     DBX 105.0;	//->"BinDB".PCRead.Status.StaLoaded
      AN    DBX 43.7;	// "BinDB".ToASW.InfEmptyingEnd 
      A     DBX 63.7;	// "BinDB".ToSSW.InfReleaseEmptyingTime
      =     DBX 105.1;	//-> "BinDB".PCRead.Status.StaEmptying
//  Init command
      A     DBX 60.5;	// "BinDB".VarCommand.InfBinNotInRecipe
      S     DBX 43.2;	// "BinDB".ToASW.InfDeselect
      A     DBX 63.4;	// "BinDB".ToSSW.CmdPulseTimer
      R     DBX 63.4;	//->"BinDB".ToSSW.CmdPulseTimer
//Test Last Bin Active
      AN    DBX 39.7;	// "BinDB".VarTemp.Value10.Flag7              [3.0]
      O     DBX 60.6;	// "BinDB".VarCommand.InfEmptyRecipe          [3.0]
      BEC;	//                                            [2.0]
      CALL  "GCS7_BinCtrlMain" (
           CODE                     := 18);	// Test Recipe/ Test Last Bin Active          [3.0]
      BEU;
      NOP   0;
NETWORK
TITLE =  METHODE DECODER
C1:   L     #CODE;
      L     1;
      <>I;
      JC    dEnd;
      OPN   DI [DBW 4];	// DB["BinDB".Para.ParSecDB]
      L     DIW 4;	// "SecDB".Para.ParLineDB
      T     #VarLineDB;	//   
      OPN   DI [#VarLineDB];	// OPN LineDB
      AN    DIX 145.0;	// "LineDB".JobWrite.Hsk.F_Define
      AN    DIX 145.1;	// "LineDB".JobWrite.Hsk.F_Execute
      AN    DIX 145.2;	// "LineDB".JobWrite.Hsk.F_Modify
      R     DBX 60.6;	// "BinDB".VarCommand.InfEmptyRecipe [1.6]
      BEC;	// 
      L     DBW 2;	//  "BinDB".Para.ParObjNr
      T     DIW 20;	//  "LineDB".VarTemp[1]= VAR_BLOCK_NR
      CDB;
      CALL  "GCS7_LineCtrlSub" (
           CODE                     := 1);	//   Line.Subroutine BlockAdr
      CDB;
      L     0;	//  
      L     DIW 22;	//  "LineDB".VarTemp[2]=VarByteNr
      ==I;	//    
      BEC;	//  --> not datas for bin
      T     #VarInByteRecipe;
      T     DBW 22;	//  "LineDB".VarTemp[2] = VarByteNr recipe
      L     #VarLineDB;
      T     DBW 20;	//  "BinDB".VarTemp.InValue= InpDBSourceRecipe
      CALL  "GCS7_BinCtrlSub" (
           CODE                     := 1);	//  Subroutine TestRecipe
      L     0;	//    
      L     DBW 36;	//  VarTemp.Value9=out_error_bin
      <>I;	// 
      JC    dErr;	// 
      L     DBW 16;	// BIN.ParNrOfBytePerIngr
      L     DBW 18;	// BIN.ParNrOfIngr
      *I;	// 
      +     6;	// 
      T     #VarLenRecipe;	// --> LENGTH RECIPE
      A     DBX 39.3;	// "BinDB".VarTemp.Value10.tmpEmptyRecipe
      =     DBX 60.6;	// "BinDB".VarCommand.InfEmptyRecipe
      OPN   DI [#VarLineDB];
      OPN   DI [DIW 4];	//-->CALL SECTION-DB DB["LineDB".Para.ParFirstSecDB]
//   ==== START LOOP SECTION =====
dLOP: L     DINO;
      T     #VarSecDB;
      AN    DIX 44.7;	// "SecDB".ToASW.InfSameJobLineDB
      JC    dNxt;	// 
      CALL  "SYS_Copy_DBtoDB" (
           DBSource                 := #VarLineDB,
           ByteSource               := #VarInByteRecipe,
           DBDest                   := #VarSecDB,
           ByteDest                 := DBW 14,
           NoOfByte                 := #VarLenRecipe,
           Fault                    := #VarError);	// "BinDB".Para.ParByteRecipeMemory
dNxt: L     DIW 8;	// "SecDB".Para.ParNextSecDB
      L     0;	// 
      ==I;	// no next section
      JC    dINI;	// 
      OPN   DI [DIW 8];	// ->CALL SECTION-DB["SecDB".Para.ParNextSecDB]
      JU    dLOP;
// ===== END LOOP SECTION ========
dINI: OPN   DI [DBW 4];	//  DB[Bin.ParSecDB ]
      A     DIX 44.7;	// "SecDB".ToASW.InfSameJobLineDB
      S     DBX 42.7;	// "BinDB".ToASW.CmdNewData
      S     DBX 60.7;	// "BinDB".VarCommand.CmdNewValue (SSW)
      A     DBX 60.7;	// "BinDB".VarCommand.CmdNewValue (SSW)
      AN    DBX 43.0;	//  "BinDB".ToASW.InfActive
      S     DBX 61.0;	// "BinDB".VarCommand.CmdFirst
      OPN   DI [#VarLineDB];	// CALL LineDB
      L     DBW 2;	// "BinDB".Para.ParObjNr 
      T     DIW 20;	// "LineDB".VarTemp[1] =VAR_OBJEKT_NR
      CDB;
      CALL  "GCS7_LineCtrlSub" (
           CODE                     := 2);	// Soubrotine ResetObjMask
      BEU;
//   ========= error code =========
dErr: OPN   DI [#VarLineDB];	// CALL LineDB
      T     DIW 138;	// "LineDB".JobRead.ErrElement
      L     30;	// 
      T     DIW 140;	// "LineDB".JobRead.ErrCode
      L     DBW 2;	// "BinDB".Para.ParObjNr
      T     DIW 142;	// "LineDB".JobRead.ErrObject
      BEU;
dEnd: NOP   0;
NETWORK
TITLE =  METHODE Init_Data
      L     #CODE;
      L     2;
      <>I;
      JC    eEnd;
      CALL  "GCS7_BinCtrlMain" (
           CODE                     := 18);	// Test Recipe/ Test Last Bin Active
      SET;
      S     DBX 43.3;
      S     DBX 43.6;	// "BinDB".ToASW.OutJobChange [2.0]
      R     DBX 105.3;	// "BinDB".PCRead.Status.StaRegistrated    [3.0]
      R     DBX 62.1;	// "BinDB".ToSSW.CmdSendResult       [3.0]
      R     DBX 82.1;	// "BinDB".PCWrite.Hsk.Q_Result      [3.0]
      R     DBX 94.1;	// "BinDB".PCRead.Hsk.F_Result       [3.0]
      CALL  "GCS7_BinCtrlSub" (
           CODE                     := 6);	// Subroutine Clear Value
      OPN   DI [DBW 4];	// CALL DI"BinDB".Para.ParSecDB]
      L     DBD 106;	// "BinDB".PCRead.JobNr
      L     DID 160;	// "SecDB".JobNom.JobNr
      T     DBD 106;	// "BinDB".PCRead.JobNr
      <>D;	// 
      O(;	// 
      L     DIW 206;	// "SecDB".JobAc.BatchNo
      T     DBW 110;	// "BinDB".PCRead.BatchNr
      L     1;	//  
      <=I;	// 
      );	// 
      ON    DBX 43.0;	// "BinDB".ToASW.InfActive [3.3]
      =     #VarNewJob;
      L     0;	// 
      T     DBD 44;	// -> "BinDB".ToASW.VarTaraWeight
      T     DBD 64;	// -> "BinDB".ToSSW.WeightTotal
      A     DBX 7.0;	// "BinDB".Para.ParTypeDef.ParBlend 
      JC    eBLD;
//   ===== TRANSPORT ===============
      AN    #VarNewJob;
      S     DBX 60.7;	// "BinDB".VarCommand.CmdNewValue 
      BEC;
      CALL  "GCS7_BinCtrlSub" (
           CODE                     := 4);	//   Subroutine Deselect all
//  [2A -->
      SET;	//   
      R     DBX 38.7;	//   var_second_loop 
//   <-- 2A]
F1:   CALL  "GCS7_BinCtrlSub" (
           CODE                     := 11);	//   Subroutine Read First
      A     DBX 39.0;	//  "BinDB".VarTemp.Value10.tmpBinNotFound1
      JC    eErr;	//  
      L     DBW 20;	// "BinDB".VarTemp.InValue=OutBinNr
      T     DBW 50;	// "BinDB".ToASW.BinPreselected 
      CALL  "GCS7_BinCtrlSub" (
           CODE                     := 2);	//   Subroutine ReadBin
      A     DBX 39.0;	// "BinDB".VarTemp.Value10.tmpBinNotFound1 
      JC    eErr;
//  [2A -->
      AN    DBX 24.0;	// "BinDB".VarTemp.Bin.InfLocked
      AN    DBX 24.1;	//"BinDB".VarTemp.Bin.InfLevelFault
      O     DBX 38.7;	// var_second_loop 
      JC    T_SE;
      S     DBX 38.7;	// var_second_loop 
FNxt: CALL  "GCS7_BinCtrlSub" (
           CODE                     := 12);	// Subroutine Read Next
      A     DBX 39.0;	// "BinDB".VarTemp.Value10.tmpBinNotFound1
      JC    F1;
      L     DBW 20;	// "BinDB".VarTemp.InValue=OutBinNr
      T     DBW 50;	// "BinDB".ToASW.BinPreselected
      CALL  "GCS7_BinCtrlSub" (
           CODE                     := 2);	// Subroutine ReadBin
      A     DBX 39.0;	//  "BinDB".VarTemp.Value10.tmpBinNotFound1 
      JC    F1;	//   [2.1]
//        SPB   eErr                      //   [2.1]
      A     DBX 24.0;	// "BinDB".VarTemp.Bin.InfLocked 
      O     DBX 24.1;	// "BinDB".VarTemp.Bin.InfLevelFault
      JC    FNxt;	//   [2.1]
//      SPB   F1                          //   [2.1]
//   <-- 2A]
T_SE: AN    DBX 25.0;	// "BinDB".VarTemp.Bin.InfActiveBin [1D]
      O     DBX 25.2;	// "BinDB".VarTemp.Bin.InfDeselect
      S     DBX 25.1;	// "BinDB".VarTemp.Bin.InfPreselect
      R     DBX 25.2;	// "BinDB".VarTemp.Bin.InfDeselect 
      A     DBX 25.0;	// "BinDB".VarTemp.Bin.InfActiveBin [1.7]
      R     DBX 25.1;	// "BinDB".VarTemp.Bin.InfPreselect  [1.7]
      CALL  "GCS7_BinCtrlSub" (
           CODE                     := 3);	// Subroutine Store Bin
      L     2#10;	// CODE= Read Value
      T     DBW 20;	// "BinDB".VarTemp.InValue   
      CALL  "GCS7_BinCtrlSub" (
           CODE                     := 13);	// Subroutine Read Blend Recipe
      CALL  "GCS7_BinCtrlSub" (
           CODE                     := 0);	//   Subroutine Test Bin Status
      BEU;
//   ==== BLEND RECIPE =============
eBLD: CALL  "GCS7_BinCtrlSub" (
           CODE                     := 4);	// Subroutine Deslect all
      L     2#1;	// CODE= Preselect
      T     DBW 20;	// "BinDB".VarTemp.InValue 
      CALL  "GCS7_BinCtrlSub" (
           CODE                     := 13);	// Subroutine Read Blend Recipe
      CALL  "GCS7_BinCtrlSub" (
           CODE                     := 0);	// Subroutine Test Bin Status
      L     2#10;	// CODE= Read Value
      T     DBW 20;	// "BinDB".VarTemp.InValue 
      AN    DBX 43.1;	// "BinDB".ToASW.InfPreselect
      AN    DBX 43.2;	// "BinDB".ToASW.InfDeselect 
      JCN   eX05;
      CALL  "GCS7_BinCtrlSub" (
           CODE                     := 13);	// Subroutine Read Blend Recipe
      CALL  "GCS7_BinCtrlSub" (
           CODE                     := 0);	// Subroutine Test Bin Status
eX05: NOP   0;
eErr: BEU;
//  =====ERROR ====================
eEnd: NOP   0;
NETWORK
TITLE =  Methode O_BIN (Code=7)
      L     #CODE;
      L     7;
      <>I;
      JC    fEnd;
      L     DBW 82;	//  "BinDB".PCWrite.Hsk
      L     0;
      ==I;
      BEC;
//-- commands --------------
      AN    DBX 83.0;	// "BinDB".PCWrite.Hsk.F_Define
      JC    Q9;
      L     0;
      T     DBW 96;	// "BinDB".PCRead.ErrElement
      T     DBW 98;	// "BinDB".PCRead.ErrCode 
      A     DBX 85.0;	// "BinDB".PCWrite.Func.CmdFirst
      S     DBX 61.0;	// "BinDB".VarCommand.CmdFirst 
      A     DBX 85.1;	// "BinDB".PCWrite.Func.CmdNext
      S     DBX 61.1;	// "BinDB".VarCommand.CmdNext
Q9:   A     DBX 82.1;	//  "BinDB".PCWrite.Hsk.Q_Result
      S     DBX 105.3;	//  "BinDB".PCRead.Status.StaRegistrated
      A     DBX 82.2;	//  "BinDB".PCWrite.Hsk.Q_ResultPrev
      S     DBX 105.6;	//  "BinDB".PCRead.Status.StaRegistratedPrev
      L     DBW 82;	// "BinDB".PCWrite.Hsk
      INVI;	//   
      L     DBW 94;	// "BinDB".PCRead.Hsk.F_xxx
      AW;	// 
      T     DBW 94;	// "BinDB".PCRead.Hsk.F_xxx
      S     DBX 41.1;	// "BinDB".ChangeBit.CBit2 (Write interface free)
      L     0;	//    
      T     DBW 82;	// "BinDB".PCWrite.Hsk
//      L     DBW   94                    // "BinDB".PCRead.Hsk
//      <>I                               //   
//      BEB                               //  
//      T     DBW   98                    // "BinDB".PCRead.ErrCode 
      BEU;	//   
fEnd: NOP   0;
NETWORK
TITLE =  Methode Test Recipe
      L     #CODE;	//   )
      L     8;	//   )  CODE= KF+8
      <>I;	//   )
      JC    gEnd;	//   )
      L     DBW 14;	// "BinDB".Para.ParByteRecipeMemory
      T     DBW 22;	//  "BinDB".VarTemp.Bin.BinNrByteNr (source_recipe)
      CALL  "GCS7_BinCtrlSub" (
           CODE                     := 1);	//   Call Subroutine Test Recipe
      BEU;
gEnd: NOP   0;
NETWORK
TITLE =  Methode Test Recipe: Test Last Ingredient active
      L     #CODE;	//   )
      L     18;	//   )  CODE= KF+8
      <>I;	//   )
      JC    jEnd;	//   )
      L     DBW 4;	// "BinDB".Para.ParSecDB
      T     DBW 20;	//-> "BinDB".VarTemp.InValue = InpDBSourceRecipe
      L     DBW 14;	// "BinDB".Para.ParByteRecipeMemory
      T     DBW 22;	//->"BinDB".VarTemp[2] = VarByteNr recipe
      CALL  "GCS7_BinCtrlSub" (
           CODE                     := 1);	//      Subroutine TestRecipe
      A     DBX 39.3;	//   <-- "BinDB".VarTemp10.tmpEmptyRecipe
      =     DBX 60.6;	//   -->"BinDB".VarCommand.InfEmptyRecipe
      L     DBW 26;	//-->Number availabel ingredient     [2.0]
      L     1;
      <=I;
      =     DBX 104.0;	// "BinDB".PCRead.Status.StaLastBinActive
      BEU;
jEnd: NOP   0;
NETWORK
TITLE = Metothe TOTALIZER (Code=10)
//Input:
//Output:
//  DBD64    0            // "BinDB".ToSSW.WeightTotal
//
      L     #CODE;
      L     10;
      <>I;
      JC    kEnd;
//Start Adress Loop
      L     DBW 8;	//"BinDB".Para.ParByteFirstBin
      SLD   3;
      LAR1;	//-->Pointer 1st Bin
// (--loop bin: test  ----------)
      L     0;
      T     DBD 64;
      L     DBW 12;	//  "BinDB".Para.ParNoOfBin
      ==I;
      JC    kFER;
kLop: T     #VarCnt;
      L     DBD [AR1,P#6.0];	// binlist[n].Bin.WeightActual
      L     DBD 64;
      +D;
      T     DBD 64;
      L     #VarLenBinBit;
      +AR1;
      L     #VarCnt;
      LOOP  kLop;
//  (--END LOOP TEST -----------)
kFER: BEU;
kEnd: NOP   0;
NETWORK
TITLE = Methode JobChange (Code=11)
//Input:
//Output:
//  DBD64    0            // "BinDB".ToSSW.WeightTotal
//
      L     #CODE;
      L     11;
      <>I;
      JC    mEnd;
//Start Adress Loop
      L     DBD 106;	//"BinDB".PCRead.JobNr 
      T     DBD 124;	//"BinDB".PCRead.JobNrPrev 
      L     DBW 110;	//"BinDB".PCRead.BatchNr 
      T     DBW 128;	//"BinDB".PCRead.BatchNrPrev 
      L     DBW 8;	//"BinDB".Para.ParByteFirstBin
      SLD   3;
      LAR1;	//-->Pointer 1st Bin
      L     DBW 10;	// "BinDB".Para.ParNoOfBytePerBin
      L     18;
      <I;
      JC    mRes;
// (--loop bin: test  ----------)
      L     0;
      L     DBW 12;	//  "BinDB".Para.ParNoOfBin
      ==I;
      JC    mRes;
mLop: T     #VarCnt;
      L     DBD [AR1,P#6.0];	// binlist[n].Bin.WeightActual
      T     DBD [AR1,P#14.0];	// binlist[n].Bin.WeightActualPrev
      L     #VarLenBinBit;
      +AR1;
      L     #VarCnt;
      LOOP  mLop;
//  (--END LOOP TEST -----------)
mRes: AN    DBX 94.2;	// "BinDB".PCRead.Hsk.F_ResultPrev
      AN    DBX 105.3;	// "BinDB".PCRead.Status.StaRegistrated
      R     DBX 105.6;	// "BinDB".PCRead.Status.StaRegistratedPrev
      S     DBX 94.2;	// "BinDB".PCRead.Hsk.F_ResultPrev 
      R     DBX 82.2;	// "BinDB".PCWrite.Hsk.Q_ResultPrev
      S     DBX 41.0;	// "BinDB".ChangeBit.CBit1      [3.1]
      BEU;
mEnd: NOP   0;
NETWORK
TITLE =  METHODE  21/22: Add Ingredient
//Code=21: Add First
//Code=22: Add Special Bin 
//
//Input Parameter: "BinDB".VarTemp.Bin.BinNrByteNr (DBW22) = Bin-Nr Ingredient
      L     21;	//Add First
      L     #CODE;
      <>I;
      A(;
      L     22;	//Add Special Bin  = Last Ingr
      <>I;
      );
      JC    igEn;
      A     DBX 7.0;	// "BinDB".Para.ParTypeDef.ParBlend 
      BEC;	//Not Suported for blend
      OPN   DI [DBW 4];	// DB["BinDB".Para.ParSecDB]
      L     DIW 4;	// "SecDB".Para.ParLineDB
      T     #VarLineDB;	//   
      OPN   DI [#VarLineDB];	// OPN LineDB
      L     DBW 2;	//  "BinDB".Para.ParObjNr
      T     DIW 20;	//  "LineDB".VarTemp[1]= VAR_BLOCK_NR
      CDB;
      CALL  "GCS7_LineCtrlSub" (
           CODE                     := 1);	//   Line.Subroutine BlockAdr
      CDB;
      L     0;	//  
      L     DIW 22;	//  "LineDB".VarTemp[2]=VarByteNr
      ==I;	//    
      BEC;	//  --> not datas for bin
      T     #VarInByteRecipe;
      L     21;	//Add First
      L     #CODE;
      ==I;
      L     1;
      JC    igSt;
      L     DBW 18;	// BIN.ParNrOfIngr
igSt: +     -1;
      T     #VarIngrIdx;
      L     0;
      <I;
      BEC;
      L     DBW 16;	// BIN.ParNrOfBytePerIngr
      L     #VarIngrIdx;
      *I;	// 
      +     L#6;	// Header
      SLD   3;
      LAR1;	//--> Pointer to Ingredient
      L     DBW 22;	//"Header".VarTemp.Bin.BinNrByteNr
      T     DBW [AR1,P#0.0];
      BEU;
igEn: NOP   0;
END_FUNCTION

